	(*****Estop*****)
	IF NOT bEstop  THEN	
		IF eState <> E_Station.eAborted AND eState <> E_Station.eAborting AND eState <> E_Station.eDisabled THEN
				eState 				:= E_Station.eAborting; 
		END_IF
	END_IF
	
	IF bEstop AND bEmergencyUp THEN
		eState 				:= E_Station.eAborting;
	END_IF

	
	CASE eState OF
	/////////////////////////////	
		E_Station.eDisabled: 					// Stan nieaktywnosci (Stacja wyłączona) 
		
			IF bEnable THEN
				eState 				:= E_Station.ePreparingToReady; 
			END_IF 
			
    /////////////////////////////	    
		E_Station.eAborted: 					// Stan bezpiecznego zatrzymania (po Abortingu) 

			IF bEStop THEN
				eState 				:= E_Station.ePreparingToReady;
			END_IF
			
	/////////////////////////////	
		E_Station.eAborting:                 	// Stan bezpiecznego zatrzymywania (po EStopie)
			IF NOT bEstop THEN 
				bBlockActuator 			:= FALSE;
				bLidSealingActuator		:=	FALSE;
				bHeightMotorDown		:=	FALSE;
				bHeightMotorUp			:=	FALSE;
				eState 					:=	E_Station.eAborted;  
				eRunningState			:=	E_LidSealing.eDisabled;
				
			ELSIF bEmergencyUp THEN
								
				bHeightMotorUp			:= NOT tofHeightMotorDown.Q ;
				bHeightMotorDown		:= FALSE;
				bLidSealingActuator		:= FALSE;
				bHomingDone 			:= FALSE;
				IF tonHeightNoChange.Q THEN	
					bHeightMotorEncoderCounterReset	:= TRUE;
					bHeightMotorUp					:= FALSE;
   				END_IF
				
			END_IF
		 
	/////////////////////////////			
		E_Station.eError:                 	 	// Stan błędu 	
			bBlockActuator := FALSE;
			IF bReset THEN
				eState 				:= E_Station.eResetting;
				
			END_IF
			
	/////////////////////////////
		E_Station.eResetting:					// Stan resetowania bledu (po Errorze)
			
			bError := FALSE;
			IF NOT bError THEN
				nErrorNr 			:=	0;
   				sErrorDescription 	:=	'';
				sErrorDescription2	:=	'';
				bTempRegulatorReset := FALSE;
				eState 				:=	E_Station.ePreparingToReady;
			ELSE
				eState 				:=	E_Station.eError;
			END_IF
        
	/////////////////////////////
		E_Station.eManualMovement:     			// Stan ruchów manualnych  
       
			ManualMovements();
			//Wyjście z trybu serwisowego
			IF NOT bManualMovement THEN
				bLidSealingActuator			:=	FALSE;
				bHeightMotorUp				:=	FALSE;
				bHeightMotorDown			:=	FALSE;
				bManualLidSealingActuator	:=	bLidSealingActuator;
				eState:=E_Station.eReady;
			END_IF

	/////////////////////////////
		E_Station.eHoming:						// Stan bazowania 

			Homing();
			IF NOT bHoming AND NOT bHeightSet THEN
			   	eState:=E_Station.ePreparingToReady;
			  	bHeightMotorDown:=FALSE;
				bHeightMotorUp:=FALSE;
			END_IF		
			
	/////////////////////////////
		E_Station.eHomingDone:                  // Stan wykonania bazowania 
		
			bHeightMotorDown					:=	FALSE;
			bHeightMotorUp						:=	FALSE;
			bHeightMotorEncoderCounterReset		:=	FALSE;
			bHomingDone							:=	TRUE;
			IF NOT bHoming AND NOT bHeightSet THEN
			  	 eState:=E_Station.eReady;
			END_IF
			
	/////////////////////////////
		E_Station.ePreparingToReady:            // Stan przygotowywania do gotowosci (zawsze przed Ready)  
		
         	bLidSealingActuator:=FALSE;
			eRunningState:=E_LidSealing.eReady;
			eState:=E_Station.eReady;	
			
	/////////////////////////////
		E_Station.ePreparingToDisable:          // Stan przygotowywania do nieaktywnosci (po wyłączeniu Enable) 
  
			bLidSealingActuator:=FALSE;
			
			bHeightMotorUp:=TRUE;
			bHeightMotorDown:=FALSE;	
			IF tonHeightNoChange.Q THEN
				bHeightMotorUp:=FALSE;
				eState:=E_Station.eDisabled;
				eRunningState:=E_LidSealing.eDisabled;
			END_IF	
			
			
	/////////////////////////////
		E_Station.eReady:						// Stan gotowosci 
		
			IF bRun AND NOT bCycleDone AND NOT bCycleNotDone THEN
				eState 				:= E_Station.eStarting; 
			END_IF
			IF bHoming OR bHeightSet THEN
				eState 				:= E_Station.eHoming; 
			END_IF
			IF bManualMovement THEN
				//Jeśli przejście w tryb ruchów manualnych przepisz wszystkie stany siłowników sterowanych przez moduł
				//aby zapobiec ewentualnym kolizjom po wejściu w tryb serwisowy
				bManualLidSealingActuator	:= bLidSealingActuator;
				bManualHeightMotorUp		:= bHeightMotorUp;
				bManualHeightMotorDown		:= bHeightMotorDown;
				bBlockActuator				:= FALSE;
				eState 						:= E_Station.eManualMovement; 
			END_IF
			IF NOT bRun THEN
				bCycleDone 					:= FALSE;
				bCycleNotDone 				:= FALSE;			
			END_IF
			
	/////////////////////////////
		E_Station.eStopping:					// Stan zatrzymywania 
			
			Running();
			eState 					:= E_Station.eReady;	
			
	/////////////////////////////
		E_Station.eStarting:                  	// Stan uruchamiania (po Ready)
		
			eState					 := E_Station.eRunning; 
			
	/////////////////////////////
		E_Station.eRunning:               		// Stan wykonywania cyklu (po Startingu), w tym stanie osobny
 
			Running();
			IF NOT bRun THEN					(*Przerywanie cyklu*)
				eState 				 := E_Station.eStopping;	
			END_IF
			IF bCycleDone OR bCycleNotDone THEN (*Cykl zakończony*)
				eState 				 := E_Station.eReady;
			END_IF	
			
	/////////////////////////////		
	END_CASE
END_ACTION

ACTION EncoderTest:


rtbHeightMotorEncoderPulse(CLK:=bHeightMotorEncoderPulse,Q=>);
ftbHeightMotorEncoderPulse(CLK:=bHeightMotorEncoderPulse,Q=>);


IF rtbHeightMotorEncoderPulse.Q THEN
	lrHeightMotorEncoderPulses	:=	lrHeightMotorEncoderPulses +	1;
END_IF
END_ACTION

ACTION ErrorHandling:
//OBSŁUGA BŁĘDÓW
// Alarm_0380	380	Error	Blokada siłownika podczas podnoszenia - sprawdź czujnik
// Alarm_0381	381	Error	Blokada siłownika podczas opuszczania - sprawdź czujnik
// Alarm_0382	382	Error	Błąd czujnika temperatury grzałki - sprawdź połączenie
// Alarm_0383	383	Error	Blokada podnośnika lub brak zasilania - sprawdź czujnik lub odblokuj mechanicznie
// Alarm_0384	384	Error	Wartość zadana wysokości jest większa od maksymalnej - zmień ustawienia w recepturze
// Alarm_0385	385	Error	Wartość zadana wysokości jest mniejsza od minimalnej - zmień ustawienia w recepturze
// Alarm_0386	386	Error	Błąd grzania, brak wzrostu temperatury - sprawdź czujnik
// Alarm_0387	387	Error	Błąd grzania, brak sygnału z czujnika temperatury - sprawdź czujnik

IF bAlarmInit THEN
    bAlarmInit := FALSE; 
	fbSourceInfo.Clear();
	fbSourceInfo.sName:=sStationName;//'Machine';
	fbSourceInfo.nId:=udiStationID;//2700;
	// Alarm_0380	380	Error	Blokada siłownika podczas podnoszenia - sprawdź czujnik
    arfbAlarm[0].CreateEx(stEventEntry := TC_EVENTS.AlarmClass.Alarm_0380, bWithConfirmation:= FALSE,  ipSourceInfo:= fbSourceInfo); 
	// Alarm_0381	381	Error	Blokada siłownika podczas opuszczania - sprawdź czujnik
	arfbAlarm[1].CreateEx(stEventEntry := TC_EVENTS.AlarmClass.Alarm_0381, bWithConfirmation:= FALSE,  ipSourceInfo:= fbSourceInfo); 
	// Alarm_0382	382	Error	Błąd czujnika temperatury grzałki - sprawdź połączenie
	arfbAlarm[2].CreateEx(stEventEntry := TC_EVENTS.AlarmClass.Alarm_0382, bWithConfirmation:= FALSE,  ipSourceInfo:= fbSourceInfo); 
	// Alarm_0383	383	Error	Blokada podnośnika lub brak zasilania - sprawdź czujnik lub odblokuj mechanicznie
	arfbAlarm[3].CreateEx(stEventEntry := TC_EVENTS.AlarmClass.Alarm_0383, bWithConfirmation:= FALSE,  ipSourceInfo:= fbSourceInfo); 
	// Alarm_0384	384	Error	Wartość zadana wysokości jest większa od maksymalnej - zmień ustawienia w recepturze
	arfbAlarm[4].CreateEx(stEventEntry := TC_EVENTS.AlarmClass.Alarm_0384, bWithConfirmation:= FALSE,  ipSourceInfo:= fbSourceInfo); 
	// Alarm_0385	385	Error	Wartość zadana wysokości jest mniejsza od minimalnej - zmień ustawienia w recepturze
	arfbAlarm[5].CreateEx(stEventEntry := TC_EVENTS.AlarmClass.Alarm_0385, bWithConfirmation:= FALSE,  ipSourceInfo:= fbSourceInfo); 
	// Alarm_0386	386	Error	Błąd grzania, brak wzrostu temperatury - sprawdź czujnik
	arfbAlarm[6].CreateEx(stEventEntry := TC_EVENTS.AlarmClass.Alarm_0386, bWithConfirmation:= FALSE,  ipSourceInfo:= fbSourceInfo); 
	// Alarm_0387	387	Error	Błąd grzania, brak sygnału z czujnika temperatury - sprawdź czujnik
	arfbAlarm[7].CreateEx(stEventEntry := TC_EVENTS.AlarmClass.Alarm_0387, bWithConfirmation:= FALSE,  ipSourceInfo:= fbSourceInfo); 
END_IF


//GRZAŁKI NIEGOTOWE (różnica temperatury grzałki różna od zadanej +/-10 st.C 
IF (ABS(lrHeaterTemperatureCVSensor-nHeaterTemperatureSV)>nTempHisteresis AND NOT bHeaterTemperatureErrorIgnore) AND eRunningState=E_LidSealing.eReady THEN
		eRunningState:=E_LidSealing.eHeaterNotReady;		
ELSIF eRunningState=E_LidSealing.eHeaterNotReady THEN
		IF (ABS(lrHeaterTemperatureCVSensor-nHeaterTemperatureSV)<nTempHisteresis OR bHeaterTemperatureErrorIgnore) THEN
			eRunningState:=E_LidSealing.eReady;	
		END_IF	
END_IF


//************LISTA BŁĘDÓW***************
bStateError:= (eState=E_Station.eError) OR (eState=E_Station.eResetting) OR bIgnoreError;


IF bEnable THEN
	// Alarm_0380	380	Error	Blokada siłownika podczas podnoszenia - sprawdź czujnik
	//Error 1 - Zacięcie siłownika zgrzewania przy próbie podnoszenia
	tonSealingActuatorUpLag(IN:=NOT bLidSealingActuator AND NOT bLidSealingActuatorUpSensor,PT:=T#2S);
	IF tonSealingActuatorUpLag.Q THEN
		IF NOT arfbAlarm[0].bActive THEN
			bLidSealingActuator:=FALSE;
			arfbAlarm[0].Raise(nTimeStamp:=0);
		END_IF
	ELSE	
		IF  arfbAlarm[0].bActive AND bReset THEN
			arfbAlarm[0].Clear(nTimeStamp:=0, bResetConfirmation:= FALSE);
		END_IF	
// 		bLidSealingActuator:=FALSE;
// 		bError := TRUE;
// 		nErrorNr:=251;
// 		//nErrorNr := nErrorNr+iStationIndex;
// 		sErrorDescription:='Blokada siłownika podczas podnoszenia - sprawdź czujnik';
	END_IF;
	// Alarm_0381	381	Error	Blokada siłownika podczas opuszczania - sprawdź czujnik
	//Error 2 - Zacięcie siłownika zgrzewania przy próbie opuszczania
	tonSealingActuatorDownLag(IN:=bLidSealingActuator AND NOT bLidSealingActuatorDownSensor,PT:=T#2S);
	IF tonSealingActuatorDownLag.Q THEN
		IF NOT arfbAlarm[1].bActive THEN
			bLidSealingActuator:=FALSE;
			arfbAlarm[1].Raise(nTimeStamp:=0);
		END_IF
	ELSE	
		IF  arfbAlarm[1].bActive AND bReset THEN
			arfbAlarm[1].Clear(nTimeStamp:=0, bResetConfirmation:= FALSE);
		END_IF	
// 		bLidSealingActuator:=FALSE;
// 		bError := TRUE;
// 		nErrorNr:=252;
// 		//nErrorNr := nErrorNr+iStationIndex;
// 		sErrorDescription:='Blokada siłownika podczas opuszczania - sprawdź czujnik';	
	END_IF;
	// Alarm_0382	382	Error	Błąd czujnika temperatury grzałki - sprawdź połączenie
	//Error 3 - Błąd czujnika temperatury
	IF bHeaterEnable AND bTemperatureSensorFault THEN
		IF NOT arfbAlarm[2].bActive THEN
			arfbAlarm[2].Raise(nTimeStamp:=0);
			bTempRegulatorReset:=TRUE;
		END_IF
	ELSE	
		IF  arfbAlarm[2].bActive AND bReset THEN
			arfbAlarm[2].Clear(nTimeStamp:=0, bResetConfirmation:= FALSE);
		END_IF	
//		bTempRegulatorReset:=TRUE;
// 		bError := TRUE;
// 		nErrorNr:=253;
// 		//nErrorNr := nErrorNr+iStationIndex;
// 		sErrorDescription:='Błąd czujnika temperatury grzałki - sprawdź połączenie';	
	END_IF;
	// Alarm_0383	383	Error	Blokada podnośnika lub brak zasilania - sprawdź czujnik lub odblokuj mechanicznie
	//Error 4 - podnośnik nie porusza się pomimo wysterowania 
	tonErrorHeightChange(IN:=(bHeightMotorUp OR bHeightMotorDown) AND nLastPositionHeightCV=lrHeightMotorCV, PT:=T#3S);
	IF tonErrorHeightChange.Q THEN
		IF NOT arfbAlarm[3].bActive THEN
			arfbAlarm[3].Raise(nTimeStamp:=0);
			bHeightMotorUp:=FALSE;
			bHeightMotorDown:=FALSE;
		END_IF
	ELSE	
		IF  arfbAlarm[3].bActive AND bReset THEN
			arfbAlarm[3].Clear(nTimeStamp:=0, bResetConfirmation:= FALSE);
		END_IF	
// 		bHeightMotorUp:=FALSE;
// 		bHeightMotorDown:=FALSE;
// 		bError := TRUE;
// 		nErrorNr:=254;
// 		//nErrorNr := nErrorNr+iStationIndex;
// 		sErrorDescription:='Blokada podnośnika lub brak zasilania - sprawdź czujnik lub odblokuj mechanicznie';	
	END_IF
	// Alarm_0384	384	Error	Wartość zadana wysokości jest większa od maksymalnej - zmień ustawienia w recepturze
	//Error 5 - Bład nastaw max
	tonMaxHeight(IN:=nPositionHeightSV>lrMaxHeight AND NOT bHomingDone AND eState=E_Station.eReady,PT:=T#30S);
	IF tonMaxHeight.Q THEN
		arfbAlarm[4].ipArguments.Clear() .AddLReal(lrMaxHeight);
		IF NOT arfbAlarm[4].bActive THEN
			bHeightMotorUp:=FALSE;
			bHeightMotorDown:=FALSE;
			arfbAlarm[4].Raise(nTimeStamp:=0);
		END_IF
	ELSE	
		IF  arfbAlarm[4].bActive AND bReset THEN
			arfbAlarm[4].Clear(nTimeStamp:=0, bResetConfirmation:= FALSE);
		END_IF	
// 		bHeightMotorUp:=FALSE;
// 		bHeightMotorDown:=FALSE;
// 		bError := TRUE;
// 		nErrorNr:=255;
// 		//nErrorNr := nErrorNr+iStationIndex;
// 		sErrorDescription:='Wartość zadana wysokości jest większa od maksymalnej - zmień ustawienia w recepturze';
// 		sErrorDescription2:=REAL_TO_STRING(LREAL_TO_INT(lrMaxHeight));
	END_IF
	// Alarm_0385	385	Error	Wartość zadana wysokości jest mniejsza od minimalnej - zmień ustawienia w recepturze
	//Error 6 - Bład nastaw min
	tonMinHeight(IN:=nPositionHeightSV<lrMinHeight AND NOT bHomingDone AND eState=E_Station.eReady,PT:=T#30S);
	IF tonMinHeight.Q THEN
		arfbAlarm[5].ipArguments.Clear() .AddLReal(lrMinHeight);
		IF NOT arfbAlarm[5].bActive THEN
			bHeightMotorUp:=FALSE;
			bHeightMotorDown:=FALSE;
			arfbAlarm[5].Raise(nTimeStamp:=0);
		END_IF
	ELSE	
		IF  arfbAlarm[5].bActive AND bReset THEN
			arfbAlarm[5].Clear(nTimeStamp:=0, bResetConfirmation:= FALSE);
		END_IF	
// 		bHeightMotorUp:=FALSE;
// 		bHeightMotorDown:=FALSE;
// 		bError := TRUE;
// 		nErrorNr:=256;
// 		//nErrorNr := nErrorNr+iStationIndex;
// 		sErrorDescription:='Wartość zadana wysokości jest mniejsza od minimalnej - zmień ustawienia w recepturze';
// 		sErrorDescription2:=REAL_TO_STRING(LREAL_TO_INT(lrMinHeight));	
	END_IF
	// Alarm_0386	386	Error	Błąd grzania, brak wzrostu temperatury - sprawdź czujnik
	//Error 7 - Błąd czujnika temperatury
	tofbHeaterPWMOut(IN:=bHeaterPWMOut,PT:=T#30S);
	tonHeaterOnAndNotHeating(IN:=tofbHeaterPWMOut.Q AND lrHeaterTemperatureCVSensor=lrHeaterTemperatureCVSensorLast AND NOT bIgnoreError , PT:=T#5M);
	lrHeaterTemperatureCVSensorLast := lrHeaterTemperatureCVSensor;
	IF tonHeaterOnAndNotHeating.Q THEN
		IF NOT arfbAlarm[6].bActive THEN
			bTempRegulatorReset 	:= TRUE;
			arfbAlarm[6].Raise(nTimeStamp:=0);
		END_IF
	ELSE	
		IF  arfbAlarm[6].bActive AND bReset THEN
			arfbAlarm[6].Clear(nTimeStamp:=0, bResetConfirmation:= FALSE);
		END_IF	
//  		bTempRegulatorReset 	:= TRUE;
// 		bError 					:= TRUE;
// 		nErrorNr 				:= 257;
// 		//nErrorNr				:=nErrorNr+iStationIndex;
// 		sErrorDescription 		:= 'Błąd grzania, brak wzrostu temperatury - sprawdź czujnik';	
	END_IF
	// Alarm_0387	387	Error	Błąd grzania, brak sygnału z czujnika temperatury - sprawdź czujnik
	//Error 8 - Błąd czujnika temperatury, wskazuje 0
	tonHeaterOnAndSensorShows0(IN:=bHeaterPWMOut AND lrHeaterTemperatureCVSensor<1 AND NOT bIgnoreError AND NOT bStateError , PT:=T#15S);
	IF tonHeaterOnAndSensorShows0.Q THEN
		IF NOT arfbAlarm[7].bActive THEN
			bTempRegulatorReset 	:= TRUE;
			arfbAlarm[7].Raise(nTimeStamp:=0);
		END_IF
	ELSE	
		IF  arfbAlarm[7].bActive AND bReset THEN
			arfbAlarm[7].Clear(nTimeStamp:=0, bResetConfirmation:= FALSE);
		END_IF	
//  		bTempRegulatorReset 	:= TRUE;
// 		bError 					:= TRUE;
// 		nErrorNr 				:= 258;
// 		//nErrorNr				:=nErrorNr+iStationIndex;
// 		sErrorDescription 		:= 'Błąd grzania, brak sygnału z czujnika temperatury - sprawdź czujnik';	
	END_IF	
	
ELSE
	bError := FALSE;
END_IF

//*******KONIEC LISTA BŁĘDÓW***************
	

//******************PRZEJŚCIE DO eERROR*****************************

IF bError AND NOT bStateError THEN
	IF eLastState = eRunning THEN
		bCycleNotDone := TRUE;
	END_IF
	eState := E_Station.eError;
END_IF

//****************WYŚWIETLANIE STATUSU BLEDU***********************


(*Wyświetlanie błedu na wyjściu*)
bError							:= FALSE;
FOR nAlarmNumerator := 0 TO 19 DO
	bError						:= bError OR arfbAlarm[nAlarmNumerator].bActive;
END_FOR

(*Przepisywanie nazwy stacji*)
sErrorStationName:=sStationName;



//Jezeli nie zbazowane to potrzebne bazowanie
IF NOT bHeightMotorEncoderHomed  THEN
	bHomingDone:=FALSE;
END_IF
END_ACTION

ACTION HeaterRegulator:
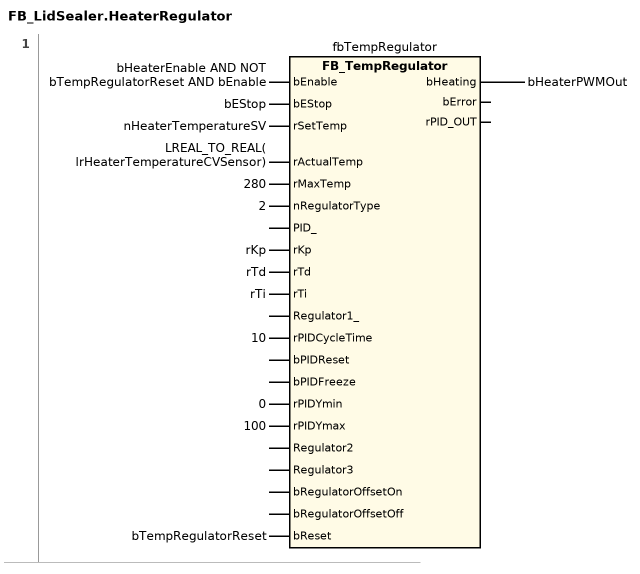
// NETWORK 1
fbTempRegulator(
    bEnable := bHeaterEnable AND NOT bTempRegulatorReset AND bEnable,
    bEStop := bEStop,
    rSetTemp := nHeaterTemperatureSV,
    rActualTemp := LREAL_TO_REAL(lrHeaterTemperatureCVSensor),
    rMaxTemp := 280,
    nRegulatorType := 2,
    rKp := rKp,
    rTd := rTd,
    rTi := rTi,
    rPIDCycleTime := 10,
    rPIDYmin := 0,
    rPIDYmax := 100,
    bReset := bTempRegulatorReset); // FB_TempRegulator
bHeaterPWMOut := fbTempRegulator.bHeating;
END_ACTION

ACTION HeightMotor:
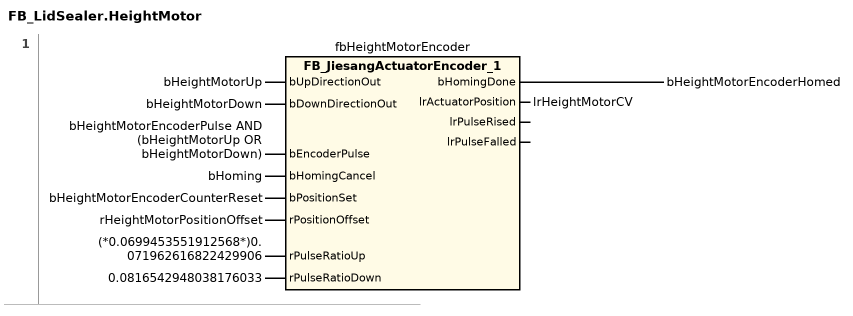
// NETWORK 1
fbHeightMotorEncoder(
    bUpDirectionOut := bHeightMotorUp,
    bDownDirectionOut := bHeightMotorDown,
    bEncoderPulse := bHeightMotorEncoderPulse AND (bHeightMotorUp OR bHeightMotorDown),
    bHomingCancel := bHoming,
    bPositionSet := bHeightMotorEncoderCounterReset,
    rPositionOffset := rHeightMotorPositionOffset,
    rPulseRatioUp := (*0.0699453551912568*)0.071962616822429906,
    rPulseRatioDown := 0.0816542948038176033,
    lrActuatorPosition => lrHeightMotorCV); // FB_JiesangActuatorEncoder_1
bHeightMotorEncoderHomed := fbHeightMotorEncoder.bHomingDone;
END_ACTION

ACTION Homing:
//BAZOWANIE
bLidSealingActuator:=FALSE;
//tofHeightMotorDown(IN:=bHeightMotorDown, PT:=T#1S); //Zabezpieczenie przed zbyt szybkim przełączeniem pomiędzy Down a Up, bezpiecznieki sie palą
		
//Podnoszenie stacji do maksymalnej pozycji
IF NOT bHeightMotorEncoderHomed OR rtEncoderHomed.Q THEN
	bHeightMotorUp:=(*TRUE*) NOT tofHeightMotorDown.Q ;
	bHeightMotorDown:=FALSE;
	IF tonHeightNoChange.Q THEN
		bHeightMotorEncoderCounterReset:=TRUE;
		bHeightMotorUp:=FALSE;
    END_IF
	//Jesli enkoder zbazowany zakończ bazowanie	
	IF rtEncoderHomed.Q THEN
		bHeightMotorUp:=FALSE;
		bHeightMotorDown:=FALSE;
		eState:=E_Station.eHomingDone;
	END_IF		
		
//Po podniesieniu stacji opuszczanie do ustalonej wysokości
ELSIF bHeightMotorEncoderHomed THEN
	bHeightMotorEncoderCounterReset:=FALSE;
	bHeightMotorUp:=lrHeightMotorCV<=nPositionHeightSV;
	bHeightMotorDown:=lrHeightMotorCV>=nPositionHeightSV;
	//Kiedy stacja osiągnie wysokość zadaną
	IF ABS(lrHeightMotorCV-nPositionHeightSV)<1 OR tonLimitPosMaxReachedDelay.Q OR tonLimitPosMinReachedDelay.Q THEN
		bHeightMotorDown:=FALSE;
		bHeightMotorUp:=FALSE;
		eState:=E_Station.eHomingDone;
	END_IF			
END_IF
END_ACTION

ACTION ManualMovements:

//W trybie ruchów manualnych wykonuj ruchy za pomocą rozkazów manualnych
IF NOT bRun THEN
	
	bBlockActuator:=bManualLidSealingActuator;
	bLidSealingActuator:=tonbBlockActuator.Q;
	bHeightMotorUp:=bManualHeightMotorUp;
	bHeightMotorDown:=bManualHeightMotorDown;
ELSE	//Kasuje zeby po cyklu nic sie nie poruszało
	bManualLidSealingActuator := FALSE;
	bManualHeightMotorUp  := FALSE;
	bManualHeightMotorDown  := FALSE;
END_IF


IF bHoming OR bHeightSet THEN
	eState:=E_Station.eHoming;
END_IF
	
Running();
	
//Zabezpieczenie przed kolizją stacji poprzez ruch podnośnika	
IF bHeightMotorDown AND lrHeightMotorCV<=lrMinHeight AND NOT bHoming AND NOT bHeightSet THEN
	bHeightMotorDown:=FALSE;
END_IF	

IF bHeightMotorUp AND lrHeightMotorCV>=lrMaxHeight AND NOT bHoming AND NOT bHeightSet THEN
	bHeightMotorUp:=FALSE;
END_IF		 

IF NOT bRun THEN
	bCycleDone 					:= FALSE;
	bCycleNotDone 				:= FALSE;	
END_IF
END_ACTION

ACTION Protections:
(*Nadpisywanie sygnałów dla bezpieczństwa mechaniki*)
IF bHeightMotorDisable THEN // Włączony siłownik blokujący podnoszenie
	bHeightMotorUp		:=FALSE;	
	bHeightMotorDown	:=FALSE;	
END_IF
END_ACTION

ACTION Running:

//Timery 
tonHeatingTime(IN:=eRunningState=E_LidSealing.eHeating,PT:=INT_TO_TIME(nLidHeatingTime));
tonbNOTLidSealingActuator(IN:=NOT bLidSealingActuator AND eRunningState=E_LidSealing.eHeating, PT:=T#100MS);
tonbBlockActuator(IN:=bBlockActuator,PT:=T#400MS);

CASE eRunningState OF
	
	//NIEGOTOWY
	E_LidSealing.eDisabled:
			eRunningState:=E_LidSealing.eReady;
		
	//ZGRZEWANIE GOTOWY DO PRACY
	E_LidSealing.eReady:
		//bLidSealingActuator:=FALSE;
		//Jeśli komenda podania platynki przejdź do stanu zasysania platynki
		IF NOT bCycleDone AND NOT bCycleNotDone THEN
			IF bRun THEN
				IF NOT bManualMovement THEN
					eRunningState:=E_LidSealing.eSealing;
				ELSE
					bBlockActuator := TRUE;
					IF tonbBlockActuator.Q THEN
						eRunningState:=E_LidSealing.eSealing;
					END_IF
				END_IF
			END_IF
		END_IF

	//STAN ZGRZEWANIA - opuszaczanie siłownika grzałki
	E_LidSealing.eSealing:
		bLidSealingActuator:=TRUE;
		//Jeśli komenda podania platynki przejdź do stanu opuszczania siłownika podajnika
		IF bLidSealingActuatorDownSensor THEN
			eRunningState:=E_LidSealing.eHeating;
		END_IF

	//ZGRZEWANIE PLATYNKI
	E_LidSealing.eHeating:
		//Zgrzewanie platynki dopóki nie osiągnie czasu przygrzewania
		IF NOT tonHeatingTime.Q THEN
			bLidSealingActuator:=TRUE;
		ELSE
			bLidSealingActuator:=FALSE;
			//IF NOT bLidSealingActuatorUpSensor THEN
			IF 	tonbNOTLidSealingActuator.Q THEN
				eRunningState:=E_LidSealing.eLidSealed;	
			END_IF
		END_IF
	
	//Zgrzewanie zakończone
	E_LidSealing.eLidSealed:
	
		bLidSealingActuator := FALSE;
		bCycleDone := TRUE;
		IF bLidSealingActuatorUpSensor THEN
			eRunningState:=E_LidSealing.eReady;
		ELSE
			eRunningState:=E_LidSealing.eGoingUp;
		END_IF

	//PODAJNIK PODNOSI SIŁOWNIK PODAWANIA PLATYNEK
	E_LidSealing.eGoingUp:
		bLidSealingActuator:=FALSE;
		bBlockActuator := FALSE;
		IF bLidSealingActuatorUpSensor THEN
			eRunningState:=E_LidSealing.eReady;
		END_IF

END_CASE
END_ACTION

ACTION Statistics:

rtrigCycleTimerRead(CLK:=(eRunningState=E_LidSealing.eLidSealed));
IF rtrigCycleTimerRead.Q THEN
		tCycleTime:=tonCycleTimer.ET;
END_IF
tonCycleTimer(IN:=eRunningState>E_LidSealing.eReady,PT:=T#1D);
END_ACTION

END_FUNCTION_BLOCK

// ---- POUs/P00_ReadRFIDCard.TcPOU
(*
Nazwa:			P00_ReadRFIDCard
Opis:			Czytnik kart zbliżeniowych
Wersja:			v0.12
Data:			2022-02-07
Autor:			DP
Urzadzenia:		
Konfiguracja:	
Info:
- Przerobienie programu na nowe czujniki RFID IFM'a
- Programować formatki trzeba po staremu bo ten bloczek IFMa nie przetestowany
*)
PROGRAM P00_ReadRFIDCard
VAR



	bReadedCardDispencer :BOOL;					(*PLC.A10*)		//Wykrycie nośnika przez czytnik przy dozownikach	
	bReadedCardBeforeScrewer :BOOL;				(*PLC.A10*)		//Wykrycie nośnika przez czytnik na 1 wjeździe karuzeli
	bReadedCardAfterScrewer :BOOL;				(*PLC.A10*)		//Wykrycie nośnika przez czytnik na 1 wjeździe karuzeli
	bReadedCardAfterDispencers :BOOL;			(*PLC.A10*)		//Wykrycie nośnika przez czytnik na 2 wjeździe karuzeli
	bReadedCardBottleTransfer :BOOL;			(*PLC.A10*)		//Wykrycie nośnika przez czytnik przy robocie
	bReadedCardCapSorter :BOOL;					(*PLC.A10*)		//Wykrycie nośnika przez czytnik przy robocie
	bReadedCardAfterDispencers2Phase :BOOL;		(*PLC.A10*)		//Wykrycie nośnika przez czytnik przy robocie
	bReadedCardLidFeeder :BOOL;					(*PLC.A10*)		//Wykrycie nośnika przez czytnik na 1 wjeździe karuzeli
	bReadedCardLidSealer :BOOL;
	
	nReadedCardDispencer :ULINT;								
	nReadedCardBeforeScrewer :ULINT;							
	nReadedCardAfterScrewer	:ULINT;
	nReadedCardAfterDispencers :ULINT;							
	nReadedCardBottleTransfer :ULINT;			
	nReadedCardCapSorter :ULINT;	
	nReadedCardAfterDispencers2Phase :ULINT;	
	nReadedCardLidFeeder :ULINT;
	nReadedCardLidSealer :ULINT;	
			
	fbWriteDataRFID: FB_WriteRFID;
	fbWriteDataRFIDnew: FB_WriteRFIDnew;
	bAutoNumber: BOOL;
	byIDtoWrite: BYTE;
	bReset: BOOL;
	bE: BOOL;
	
	(*Nowa Głowica IFM*)
	fbDispencerReader   								:   	FB_IfmIoLinkRfid;
	AusiDispencerReaderInputData  				AT%I*	: 		ARRAY[0..27] OF USINT;
	IbDispencerReaderTagPresent					AT%I*	:		BOOL;
	IBDispencerReaderErrorValue					AT%I*	:		BYTE;
	IbDispencerReaderCmdEnd						AT%I*	:		BOOL;
	IBDispencerReaderDataCounterIn				AT%I*	:		BYTE;
	IbDispencerReaderCmdStartAck				AT%I*	:		BOOL;
	IbDispencerReaderCmdStart					AT%Q*	:		BOOL;
	IBDispencerReaderCmmandValue				AT%Q*	:		BYTE;
	IBDispencerReaderDataCounterOut				AT%Q*	:		BYTE;
	AusiDispencerReaderOutputData  				AT%Q*	: 		ARRAY[0..27] OF USINT;	
	
	fbAfterDispencersReader   							:   	FB_IfmIoLinkRfid;
	AusiAfterDispencersReaderInputData  		AT%I*	: 		ARRAY[0..27] OF USINT;
	IbAfterDispencersReaderTagPresent			AT%I*	:		BOOL;
	IBAfterDispencersReaderErrorValue			AT%I*	:		BYTE;
	IbAfterDispencersReaderCmdEnd				AT%I*	:		BOOL;
	IBAfterDispencersReaderDataCounterIn		AT%I*	:		BYTE;
	IbAfterDispencersReaderCmdStartAck			AT%I*	:		BOOL;
	IbAfterDispencersReaderCmdStart				AT%Q*	:		BOOL;
	IBAfterDispencersReaderCmmandValue			AT%Q*	:		BYTE;
	IBAfterDispencersReaderDataCounterOut		AT%Q*	:		BYTE;
	AusiAfterDispencersReaderOutputData  		AT%Q*	: 		ARRAY[0..27] OF USINT;		
	ABAfterDispencersReaderWriteData					:		ARRAY[0..15] OF BYTE;

	fbLidFeederReader   								:   	FB_IfmIoLinkRfid; 	
	AusiLidFeederReaderInputData  				AT%I*	: 		ARRAY[0..27] OF USINT;
	IbLidFeederReaderTagPresent					AT%I*	:		BOOL;
	IBLidFeederReaderErrorValue					AT%I*	:		BYTE;
	IbLidFeederReaderCmdEnd						AT%I*	:		BOOL;
	IBLidFeederReaderDataCounterIn				AT%I*	:		BYTE;
	IbLidFeederReaderCmdStartAck				AT%I*	:		BOOL;
	IbLidFeederReaderCmdStart					AT%Q*	:		BOOL;
	IBLidFeederReaderCmmandValue				AT%Q*	:		BYTE;
	IBLidFeederReaderDataCounterOut				AT%Q*	:		BYTE;
	AusiLidFeederReaderOutputData  				AT%Q*	: 		ARRAY[0..27] OF USINT;		
	ABALidFeederReaderWriteData							:		ARRAY[0..15] OF BYTE;
	
	fbBeforeScrewerReader   							:   	FB_IfmIoLinkRfid;
	AusiBeforeScrewerReaderInputData  			AT%I*	: 		ARRAY[0..27] OF USINT;
	IbBeforeScrewerReaderTagPresent				AT%I*	:		BOOL;
	IBBeforeScrewerReaderErrorValue				AT%I*	:		BYTE;
	IbBeforeScrewerReaderCmdEnd					AT%I*	:		BOOL;
	IBBeforeScrewerReaderDataCounterIn			AT%I*	:		BYTE;
	IbBeforeScrewerReaderCmdStartAck			AT%I*	:		BOOL;
	IbBeforeScrewerReaderCmdStart				AT%Q*	:		BOOL;
	IBBeforeScrewerReaderCmmandValue			AT%Q*	:		BYTE;
	IBBeforeScrewerReaderDataCounterOut			AT%Q*	:		BYTE;
	AusiBeforeScrewerReaderOutputData  			AT%Q*	: 		ARRAY[0..27] OF USINT;	

	fbAfterScrewerReader   								:   	FB_IfmIoLinkRfid;
	AusiAfterScrewerReaderInputData  			AT%I*	: 		ARRAY[0..27] OF USINT;
	IbAfterScrewerReaderTagPresent				AT%I*	:		BOOL;
	IBAfterScrewerReaderErrorValue				AT%I*	:		BYTE;
	IbAfterScrewerReaderCmdEnd					AT%I*	:		BOOL;
	IBAfterScrewerReaderDataCounterIn			AT%I*	:		BYTE;
	IbAfterScrewerReaderCmdStartAck				AT%I*	:		BOOL;
	IbAfterScrewerReaderCmdStart				AT%Q*	:		BOOL;
	IBAfterScrewerReaderCmmandValue				AT%Q*	:		BYTE;
	IBAfterScrewerReaderDataCounterOut			AT%Q*	:		BYTE;
	AusiAfterScrewerReaderOutputData  			AT%Q*	: 		ARRAY[0..27] OF USINT;	

	fbBottleTransferReader   							:   	FB_IfmIoLinkRfid;
	AusiBottleTransferReaderInputData  			AT%I*	: 		ARRAY[0..27] OF USINT;
	IbBottleTransferReaderTagPresent			AT%I*	:		BOOL;
	IBBottleTransferReaderErrorValue			AT%I*	:		BYTE;
	IbBottleTransferReaderCmdEnd				AT%I*	:		BOOL;
	IBBottleTransferReaderDataCounterIn			AT%I*	:		BYTE;
	IbBottleTransferReaderCmdStartAck			AT%I*	:		BOOL;
	IbBottleTransferReaderCmdStart				AT%Q*	:		BOOL;
	IBBottleTransferReaderCmmandValue			AT%Q*	:		BYTE;
	IBBottleTransferReaderDataCounterOut		AT%Q*	:		BYTE;
	AusiBottleTransferReaderOutputData  		AT%Q*	: 		ARRAY[0..27] OF USINT;		
	
	fbCapSorterReader   								:   	FB_IfmIoLinkRfid;
	AusiCapSorterReaderInputData  				AT%I*	: 		ARRAY[0..27] OF USINT;
	IbCapSorterReaderTagPresent					AT%I*	:		BOOL;
	IBCapSorterReaderErrorValue					AT%I*	:		BYTE;
	IbCapSorterReaderCmdEnd						AT%I*	:		BOOL;
	IBCapSorterReaderDataCounterIn				AT%I*	:		BYTE;
	IbCapSorterReaderCmdStartAck				AT%I*	:		BOOL;
	IbCapSorterReaderCmdStart					AT%Q*	:		BOOL;
	IBCapSorterReaderCmmandValue				AT%Q*	:		BYTE;
	IBCapSorterReaderDataCounterOut				AT%Q*	:		BYTE;
	AusiCapSorterReaderOutputData  				AT%Q*	: 		ARRAY[0..27] OF USINT;		
	
	fbAfterDispencers2PhaseReader   						:   	FB_IfmIoLinkRfid;
	AusiAfterDispencers2PhaseReaderInputData  		AT%I*	: 		ARRAY[0..27] OF USINT;
	IbAfterDispencers2PhaseReaderTagPresent			AT%I*	:		BOOL;
	IBAfterDispencers2PhaseReaderErrorValue			AT%I*	:		BYTE;
	IbAfterDispencers2PhaseReaderCmdEnd				AT%I*	:		BOOL;
	IBAfterDispencers2PhaseReaderDataCounterIn		AT%I*	:		BYTE;
	IbAfterDispencers2PhaseReaderCmdStartAck		AT%I*	:		BOOL;
	IbAfterDispencers2PhaseReaderCmdStart			AT%Q*	:		BOOL;
	IBAfterDispencers2PhaseReaderCmmandValue		AT%Q*	:		BYTE;
	IBAfterDispencers2PhaseReaderDataCounterOut		AT%Q*	:		BYTE;
	AusiAfterDispencers2PhaseReaderOutputData  		AT%Q*	: 		ARRAY[0..27] OF USINT;		
	ABAfterDispencers2PhaseReaderWriteData					:		ARRAY[0..15] OF BYTE;
	
	fbLidSealerReader   								:   	FB_IfmIoLinkRfid; 	
	AusiLidSealerReaderInputData  				AT%I*	: 		ARRAY[0..27] OF USINT;
	IbLidSealerReaderTagPresent					AT%I*	:		BOOL;
	IBLidSealerReaderErrorValue					AT%I*	:		BYTE;
	IbLidSealerReaderCmdEnd						AT%I*	:		BOOL;
	IBLidSealerReaderDataCounterIn				AT%I*	:		BYTE;
	IbLidSealerReaderCmdStartAck				AT%I*	:		BOOL;
	IbLidSealerReaderCmdStart					AT%Q*	:		BOOL;
	IBLidSealerReaderCmmandValue				AT%Q*	:		BYTE;
	IBLidSealerReaderDataCounterOut				AT%Q*	:		BYTE;
	AusiLidSealerReaderOutputData  				AT%Q*	: 		ARRAY[0..27] OF USINT;	
	ABALidSealerReaderWriteData							:		ARRAY[0..15] OF BYTE;
	
	
	(**)
	iWriteDataCASE										:	INT;
	iWriteDataOn										:	BOOL;
	iWriteDataCount										:	INT;
	tonWriteDataCASE40									:	TON;
	
	(*RFIDCheck*)
	rtbWeighingFormDone									:	R_TRIG;

	
	tonRFIDCheckReader1Add								:	TON;
	rtRFIDCheckReader1Add								:	R_TRIG;
	tonRFIDCheckReader2Add								:	TON;
	rtRFIDCheckReader2Add								:	R_TRIG;
	tonRFIDCheckReader3Add								:	TON;
	rtRFIDCheckReader3Add								:	R_TRIG;
	tonRFIDCheckReader4Add								:	TON;
	rtRFIDCheckReader4Add								:	R_TRIG;
	tonRFIDCheckReader5Add								:	TON;
	rtRFIDCheckReader5Add								:	R_TRIG;	



	//AuliRFIDCheck										:	ARRAY [1..100] OF ULINT;	

	bRFIDCheckSave										:	BOOL;
	iRFIDCheck											:	INT;
	rtRFIDCheckbReadedCardBottleTransfer				:	R_TRIG;
	bRFIDCheckDiffrence									:	BOOL;
	iRFIDCheckProblemWithNumber							:	INT;
	sRFIDInfoSensorError								:	STRING;
	iRFIDCheckNumberOfFormsExecuteTemp					:	INT;	
	i,j													:	INT;
	
	tonRFIDCheckDispencersWarning						:	TON;
	rttonRFIDCheckDispencerWarning						:	R_TRIG;

	iRFIDCheckDispencerWarningLast						:	INT;	
	bRFIDCheckDispencerWarning							:	BOOL;
	
	tonRFIDCheckWeightWarning						:	TON;
	rttonRFIDCheckWeightWarning						:	R_TRIG;

	iRFIDCheckWeightWarningLast						:	INT;
	
	bRFIDCheckWeightWarning							:	BOOL;
	
	tonRFIDCheckBeforeScrewerWarning				:	TON;
	rttonRFIDCheckBeforeScrewerWarning				:	R_TRIG;

	iRFIDCheckBeforeScrewerWarningLast				:	INT;	
	bRFIDCheckBeforeScrewerWarning					:	BOOL;
	
	tonRFIDCheckAfterScrewerWarning					:	TON;
	rttonRFIDCheckAfterScrewerWarning				:	R_TRIG;

	iRFIDCheckAfterScrewerWarningLast				:	INT;
	
	bRFIDCheckAfterScrewerWarning					:	BOOL;	

	tonRFIDCheckBottleTransferWarning				:	TON;
	rttonRFIDCheckBottleTransferWarning				:	R_TRIG;

	iRFIDCheckBottleTransferWarningLast				:	INT;

	bRFIDCheckBottleTransferWarning					:	BOOL;	


	tonRFIDCheck10s									:	TON;
	ftRFIDCheckAfterScrewerWarning					:	F_TRIG;
	bRFIDCheckResetAll								:	BOOL;
	tonRFIDReset									:	TON;
	iRFIDReaded1Errors								: 	INT;
	iRFIDReaded2Errors								: 	INT;
	iRFIDReaded3Errors								: 	INT;
	iRFIDReaded4Errors								: 	INT;
	iRFIDReaded5Errors								: 	INT;	
	bRFIDCheckEnable								:	BOOL;
	
	(*inne*)
	




END_VAR

(*Przepisanie bity wykrycia karty*)
bReadedCardDispencer 		:= IbDispencerReaderTagPresent AND fbDispencerReader.bCodeReaded;
nReadedCardDispencer 		:= DINT_TO_ULINT(P00_ReadRFIDCard.fbDispencerReader.diReadedCode);

bReadedCardAfterDispencers 	:= IbAfterDispencersReaderTagPresent AND fbAfterDispencersReader.bCodeReaded;
nReadedCardAfterDispencers	:= DINT_TO_ULINT(P00_ReadRFIDCard.fbAfterDispencersReader.diReadedCode);

bReadedCardBeforeScrewer 	:= IbBeforeScrewerReaderTagPresent AND fbBeforeScrewerReader.bCodeReaded;
nReadedCardBeforeScrewer	:= DINT_TO_ULINT(P00_ReadRFIDCard.fbBeforeScrewerReader.diReadedCode);

bReadedCardAfterScrewer 	:= IbAfterScrewerReaderTagPresent  AND fbAfterScrewerReader.bCodeReaded;
nReadedCardAfterScrewer		:= DINT_TO_ULINT(P00_ReadRFIDCard.fbAfterScrewerReader.diReadedCode);

bReadedCardBottleTransfer 	:= IbBottleTransferReaderTagPresent AND fbBottleTransferReader.bCodeReaded;;
nReadedCardBottleTransfer	:= DINT_TO_ULINT(P00_ReadRFIDCard.fbBottleTransferReader.diReadedCode);

bReadedCardCapSorter 		:= IbCapSorterReaderTagPresent AND fbCapSorterReader.bCodeReaded;;
nReadedCardCapSorter		:= DINT_TO_ULINT(P00_ReadRFIDCard.fbCapSorterReader.diReadedCode);

bReadedCardAfterDispencers2Phase 	:= IbAfterDispencers2PhaseReaderTagPresent AND fbAfterDispencers2PhaseReader.bCodeReaded;
nReadedCardAfterDispencers2Phase	:= DINT_TO_ULINT(P00_ReadRFIDCard.fbAfterDispencers2PhaseReader.diReadedCode);

bReadedCardLidFeeder 		:= IbLidFeederReaderTagPresent AND fbLidFeederReader.bCodeReaded;;
nReadedCardLidFeeder 		:= DINT_TO_ULINT(P00_ReadRFIDCard.fbLidFeederReader.diReadedCode);

bReadedCardLidSealer 		:= IbLidSealerReaderTagPresent AND fbLidSealerReader.bCodeReaded;;
nReadedCardLidSealer 		:= DINT_TO_ULINT(P00_ReadRFIDCard.fbLidSealerReader.diReadedCode);




aIFM();
aWriteDataIFM();
aHMIShowRFID();
aRFIDCheck();
aRFIDCheckWarnings();

ACTION aHMIShowRFID:

VIS.sSlowestStation5:= Concat('RFID before scales:',ULINT_TO_STRING(nReadedCardAfterDispencers));
VIS.iSlowestStationCount5:=ULINT_TO_INT(nReadedCardAfterDispencers);
END_ACTION

ACTION aIFM:
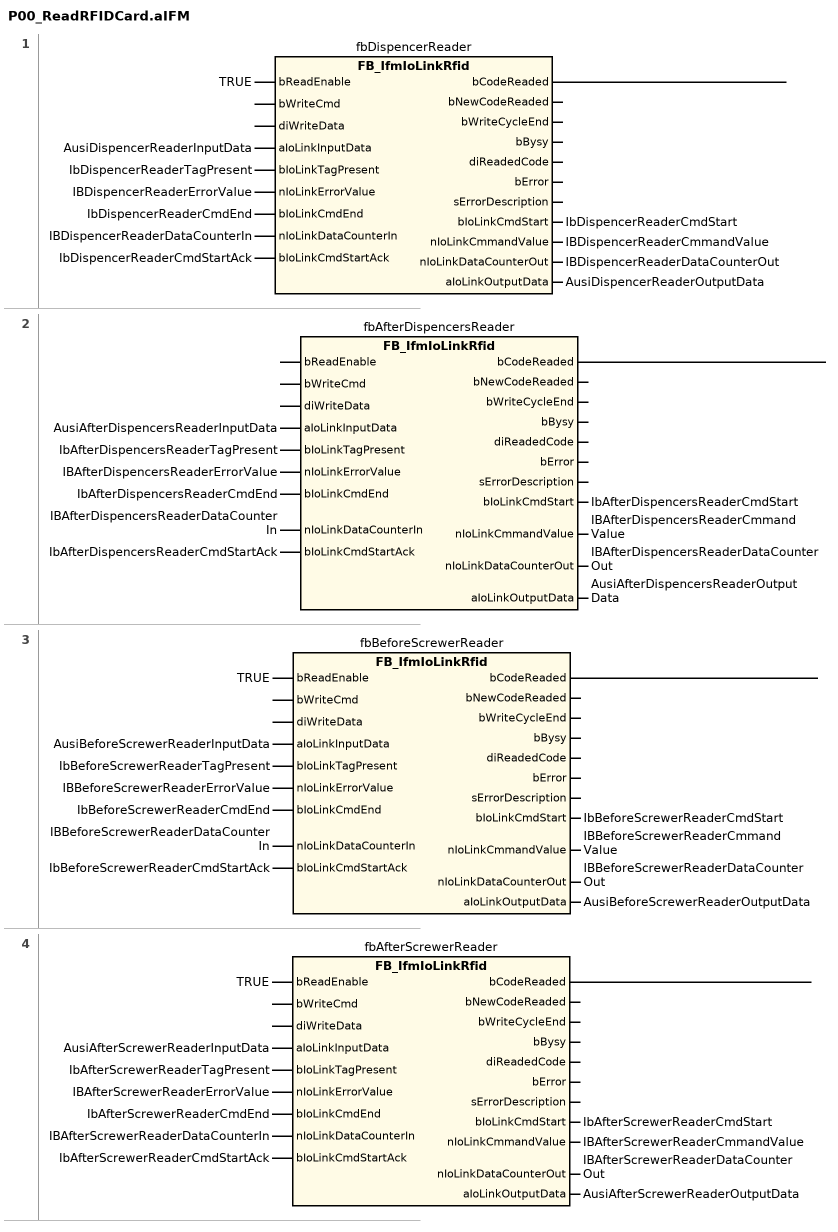
// NETWORK 1
fbDispencerReader(
    bReadEnable := TRUE,
    aIoLinkInputData := AusiDispencerReaderInputData,
    bIoLinkTagPresent := IbDispencerReaderTagPresent,
    nIoLinkErrorValue := IBDispencerReaderErrorValue,
    bIoLinkCmdEnd := IbDispencerReaderCmdEnd,
    nIoLinkDataCounterIn := IBDispencerReaderDataCounterIn,
    bIoLinkCmdStartAck := IbDispencerReaderCmdStartAck,
    bIoLinkCmdStart => IbDispencerReaderCmdStart,
    nIoLinkCmmandValue => IBDispencerReaderCmmandValue,
    nIoLinkDataCounterOut => IBDispencerReaderDataCounterOut,
    aIoLinkOutputData => AusiDispencerReaderOutputData); // FB_IfmIoLinkRfid

// NETWORK 2
fbAfterDispencersReader(
    aIoLinkInputData := AusiAfterDispencersReaderInputData,
    bIoLinkTagPresent := IbAfterDispencersReaderTagPresent,
    nIoLinkErrorValue := IBAfterDispencersReaderErrorValue,
    bIoLinkCmdEnd := IbAfterDispencersReaderCmdEnd,
    nIoLinkDataCounterIn := IBAfterDispencersReaderDataCounterIn,
    bIoLinkCmdStartAck := IbAfterDispencersReaderCmdStartAck,
    bIoLinkCmdStart => IbAfterDispencersReaderCmdStart,
    nIoLinkCmmandValue => IBAfterDispencersReaderCmmandValue,
    nIoLinkDataCounterOut => IBAfterDispencersReaderDataCounterOut,
    aIoLinkOutputData => AusiAfterDispencersReaderOutputData); // FB_IfmIoLinkRfid

// NETWORK 3
fbBeforeScrewerReader(
    bReadEnable := TRUE,
    aIoLinkInputData := AusiBeforeScrewerReaderInputData,
    bIoLinkTagPresent := IbBeforeScrewerReaderTagPresent,
    nIoLinkErrorValue := IBBeforeScrewerReaderErrorValue,
    bIoLinkCmdEnd := IbBeforeScrewerReaderCmdEnd,
    nIoLinkDataCounterIn := IBBeforeScrewerReaderDataCounterIn,
    bIoLinkCmdStartAck := IbBeforeScrewerReaderCmdStartAck,
    bIoLinkCmdStart => IbBeforeScrewerReaderCmdStart,
    nIoLinkCmmandValue => IBBeforeScrewerReaderCmmandValue,
    nIoLinkDataCounterOut => IBBeforeScrewerReaderDataCounterOut,
    aIoLinkOutputData => AusiBeforeScrewerReaderOutputData); // FB_IfmIoLinkRfid

// NETWORK 4
fbAfterScrewerReader(
    bReadEnable := TRUE,
    aIoLinkInputData := AusiAfterScrewerReaderInputData,
    bIoLinkTagPresent := IbAfterScrewerReaderTagPresent,
    nIoLinkErrorValue := IBAfterScrewerReaderErrorValue,
    bIoLinkCmdEnd := IbAfterScrewerReaderCmdEnd,
    nIoLinkDataCounterIn := IBAfterScrewerReaderDataCounterIn,
    bIoLinkCmdStartAck := IbAfterScrewerReaderCmdStartAck,
    bIoLinkCmdStart => IbAfterScrewerReaderCmdStart,
    nIoLinkCmmandValue => IBAfterScrewerReaderCmmandValue,
    nIoLinkDataCounterOut => IBAfterScrewerReaderDataCounterOut,
    aIoLinkOutputData => AusiAfterScrewerReaderOutputData); // FB_IfmIoLinkRfid

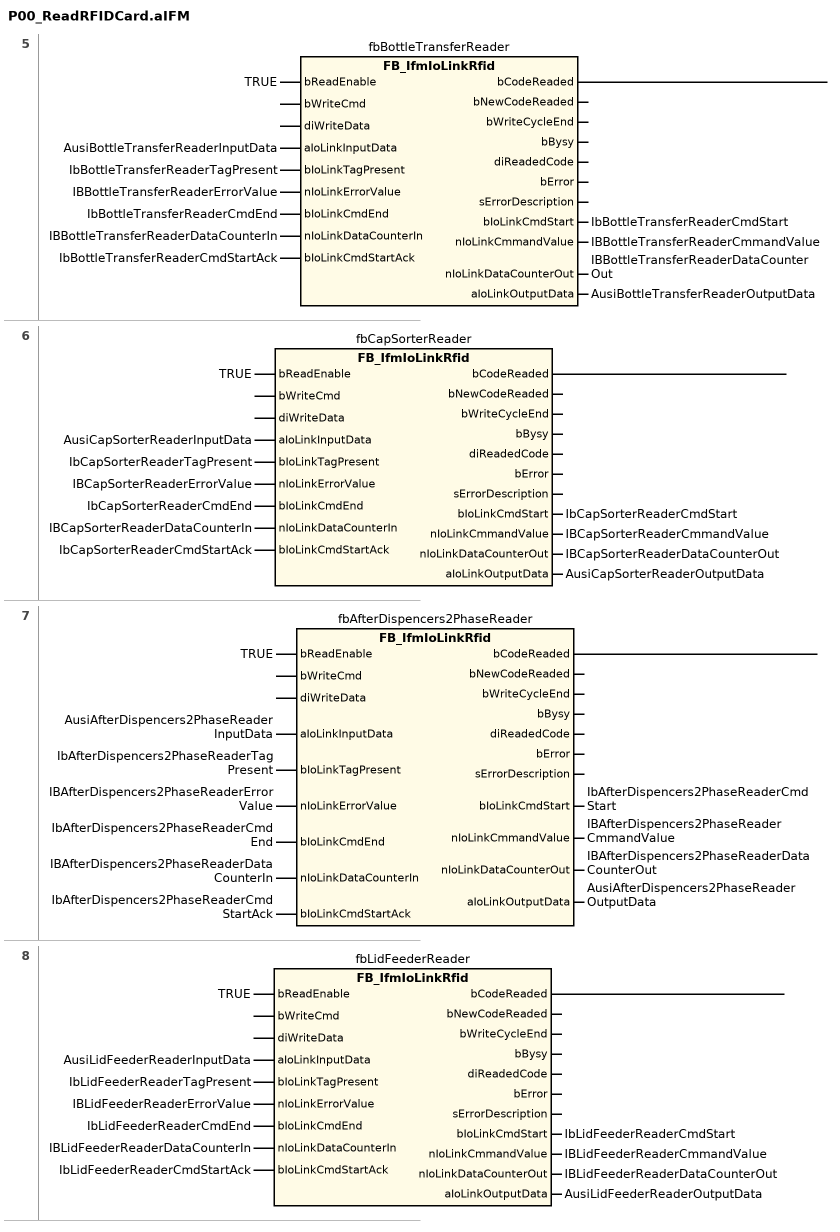
// NETWORK 5
fbBottleTransferReader(
    bReadEnable := TRUE,
    aIoLinkInputData := AusiBottleTransferReaderInputData,
    bIoLinkTagPresent := IbBottleTransferReaderTagPresent,
    nIoLinkErrorValue := IBBottleTransferReaderErrorValue,
    bIoLinkCmdEnd := IbBottleTransferReaderCmdEnd,
    nIoLinkDataCounterIn := IBBottleTransferReaderDataCounterIn,
    bIoLinkCmdStartAck := IbBottleTransferReaderCmdStartAck,
    bIoLinkCmdStart => IbBottleTransferReaderCmdStart,
    nIoLinkCmmandValue => IBBottleTransferReaderCmmandValue,
    nIoLinkDataCounterOut => IBBottleTransferReaderDataCounterOut,
    aIoLinkOutputData => AusiBottleTransferReaderOutputData); // FB_IfmIoLinkRfid

// NETWORK 6
fbCapSorterReader(
    bReadEnable := TRUE,
    aIoLinkInputData := AusiCapSorterReaderInputData,
    bIoLinkTagPresent := IbCapSorterReaderTagPresent,
    nIoLinkErrorValue := IBCapSorterReaderErrorValue,
    bIoLinkCmdEnd := IbCapSorterReaderCmdEnd,
    nIoLinkDataCounterIn := IBCapSorterReaderDataCounterIn,
    bIoLinkCmdStartAck := IbCapSorterReaderCmdStartAck,
    bIoLinkCmdStart => IbCapSorterReaderCmdStart,
    nIoLinkCmmandValue => IBCapSorterReaderCmmandValue,
    nIoLinkDataCounterOut => IBCapSorterReaderDataCounterOut,
    aIoLinkOutputData => AusiCapSorterReaderOutputData); // FB_IfmIoLinkRfid

// NETWORK 7
fbAfterDispencers2PhaseReader(
    bReadEnable := TRUE,
    aIoLinkInputData := AusiAfterDispencers2PhaseReaderInputData,
    bIoLinkTagPresent := IbAfterDispencers2PhaseReaderTagPresent,
    nIoLinkErrorValue := IBAfterDispencers2PhaseReaderErrorValue,
    bIoLinkCmdEnd := IbAfterDispencers2PhaseReaderCmdEnd,
    nIoLinkDataCounterIn := IBAfterDispencers2PhaseReaderDataCounterIn,
    bIoLinkCmdStartAck := IbAfterDispencers2PhaseReaderCmdStartAck,
    bIoLinkCmdStart => IbAfterDispencers2PhaseReaderCmdStart,
    nIoLinkCmmandValue => IBAfterDispencers2PhaseReaderCmmandValue,
    nIoLinkDataCounterOut => IBAfterDispencers2PhaseReaderDataCounterOut,
    aIoLinkOutputData => AusiAfterDispencers2PhaseReaderOutputData); // FB_IfmIoLinkRfid

// NETWORK 8
fbLidFeederReader(
    bReadEnable := TRUE,
    aIoLinkInputData := AusiLidFeederReaderInputData,
    bIoLinkTagPresent := IbLidFeederReaderTagPresent,
    nIoLinkErrorValue := IBLidFeederReaderErrorValue,
    bIoLinkCmdEnd := IbLidFeederReaderCmdEnd,
    nIoLinkDataCounterIn := IBLidFeederReaderDataCounterIn,
    bIoLinkCmdStartAck := IbLidFeederReaderCmdStartAck,
    bIoLinkCmdStart => IbLidFeederReaderCmdStart,
    nIoLinkCmmandValue => IBLidFeederReaderCmmandValue,
    nIoLinkDataCounterOut => IBLidFeederReaderDataCounterOut,
    aIoLinkOutputData => AusiLidFeederReaderOutputData); // FB_IfmIoLinkRfid

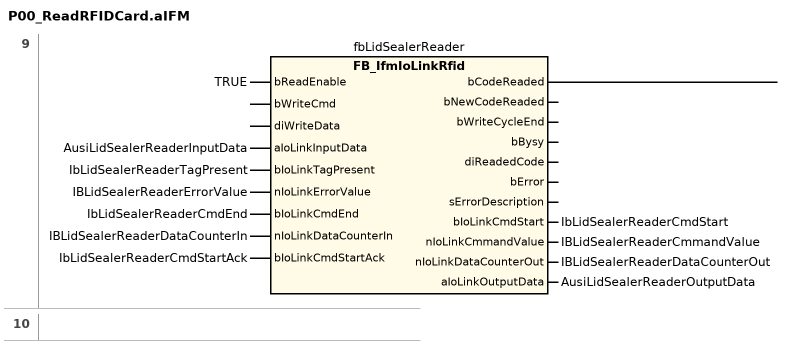
// NETWORK 9
fbLidSealerReader(
    bReadEnable := TRUE,
    aIoLinkInputData := AusiLidSealerReaderInputData,
    bIoLinkTagPresent := IbLidSealerReaderTagPresent,
    nIoLinkErrorValue := IBLidSealerReaderErrorValue,
    bIoLinkCmdEnd := IbLidSealerReaderCmdEnd,
    nIoLinkDataCounterIn := IBLidSealerReaderDataCounterIn,
    bIoLinkCmdStartAck := IbLidSealerReaderCmdStartAck,
    bIoLinkCmdStart => IbLidSealerReaderCmdStart,
    nIoLinkCmmandValue => IBLidSealerReaderCmmandValue,
    nIoLinkDataCounterOut => IBLidSealerReaderDataCounterOut,
    aIoLinkOutputData => AusiLidSealerReaderOutputData); // FB_IfmIoLinkRfid

// NETWORK 10
END_ACTION

ACTION aRFIDCheck:

//AnRFIDCardNumberShow							:ARRAY [1..100] OF ULINT;	// [H] Tabela numerów formatek 
IF VIS.AnRFIDWeightShow[1] = 0 THEN
	bRFIDCheckEnable :=	FALSE;
END_IF
rtbWeighingFormDone								(CLK:=	MAIN.bWeighingFormDone OR (NOT bFirstCycle AND VIS.AnRFIDWeightShow[1] > 0), Q=>);
IF rtbWeighingFormDone.Q THEN
	bRFIDCheckEnable :=	TRUE;
END_IF


IF bRFIDCheckResetAll THEN
	FOR i := 1 TO 100 DO												// Krok 1 - Przepisanie numerów RFID po przeważaniu
			AStRFIDCheck[i].iNumber				:=	0;
			AStRFIDCheck[i].iReaded1			:=	0;
			AStRFIDCheck[i].iReaded2			:=	0;
			AStRFIDCheck[i].iReaded3			:=	0;
			AStRFIDCheck[i].iReaded4			:=	0;
			AStRFIDCheck[i].iReaded5			:=	0;
	END_FOR		
	bRFIDCheckResetAll	:= FALSE;
END_IF

IF bRFIDCheckReset THEN
	FOR i := 1 TO 100 DO												// Krok 1 - Przepisanie numerów RFID po przeważaniu
			AStRFIDCheck[i].iReaded1			:=	0;
			AStRFIDCheck[i].iReaded2			:=	0;
			AStRFIDCheck[i].iReaded3			:=	0;
			AStRFIDCheck[i].iReaded4			:=	0;
			AStRFIDCheck[i].iReaded5			:=	0;
	END_FOR	
	
	iRFIDCheckNumberOfFormsExecute 			:= 0;
	iRFIDCheckProblemWithNumber				:= 0;
	iRFIDCheckDispencerWarning				:= 0;
	iRFIDCheckWeightWarning					:= 0;		
	iRFIDCheckBeforeScrewerWarning			:= 0;	
	iRFIDCheckAfterScrewerWarning			:= 0;	
	iRFIDCheckBottleTransferWarning			:= 0;		
	iRFIDReaded1Errors						:= 0;
	iRFIDReaded2Errors						:= 0;
	iRFIDReaded3Errors						:= 0;
	iRFIDReaded4Errors						:= 0;
	iRFIDReaded5Errors						:= 0;
	bRFIDCheckReset	:= FALSE;
END_IF


//Kasowanie w trakcie pracy i jak jest git

tonRFIDReset
	(IN:= P00_PackML.fbPMLAuto.ePMLState = Tc3_PackML.E_PMLState.ePMLState_EXECUTE AND
	iRFIDCheckDispencerWarning = iRFIDCheckDispencerWarningLast AND
	iRFIDCheckWeightWarning = iRFIDCheckWeightWarningLast AND
	iRFIDCheckBeforeScrewerWarning = iRFIDCheckBeforeScrewerWarningLast AND
	iRFIDCheckAfterScrewerWarning = iRFIDCheckAfterScrewerWarningLast AND
	iRFIDCheckBottleTransferWarning = iRFIDCheckBottleTransferWarningLast AND
	
	NOT tonRFIDReset.Q
	,PT := T#3M);

//Zapamietywanie ilości formatek po przewazaniu
IF rtbWeighingFormDone.Q OR bCycleReseting THEN	
	iRFIDCheckNumberOfFormsExecute 			:= 0;
	iRFIDCheckNumberOfFormsAfterWeighting 	:= 0;
	iRFIDCheckProblemWithNumber				:= 0;
	sRFIDInfoSensorError					:= '';
	iRFIDCheckDispencerWarning				:= 0;
	iRFIDCheckWeightWarning					:= 0;		
	iRFIDCheckBeforeScrewerWarning			:= 0;	
	iRFIDCheckAfterScrewerWarning			:= 0;	
	iRFIDCheckBottleTransferWarning			:= 0;	
	FOR i := 1 TO 100 DO												// Krok 1 - Przepisanie numerów RFID po przeważaniu
		IF VIS.AnRFIDCardNumberShow[i] > 0 THEN
			AStRFIDCheck[i].iNumber					:=	ULINT_TO_INT(VIS.AnRFIDCardNumberShow[i]);
			AStRFIDCheck[i].iReaded1				:=	0;
			AStRFIDCheck[i].iReaded2				:=	0;
			AStRFIDCheck[i].iReaded3				:=	0;
			AStRFIDCheck[i].iReaded4				:=	0;
			AStRFIDCheck[i].iReaded5				:=	0;		
			iRFIDCheckNumberOfFormsAfterWeighting	:=	iRFIDCheckNumberOfFormsAfterWeighting	+	1;
		END_IF
	END_FOR
END_IF

(*******************Reader1********************)
P00_ReadRFIDCard.bReadedCardDispencer;	nReadedCardDispencer;
tonRFIDCheckReader1Add	(IN:=	P00_ReadRFIDCard.bReadedCardDispencer,			PT:=T#10MS);
rtRFIDCheckReader1Add 	(CLK:=	tonRFIDCheckReader1Add.Q,						Q=>);
IF rtRFIDCheckReader1Add.Q AND bRFIDCheckEnable THEN
	FOR i:=1 TO 100 DO
		IF AStRFIDCheck[i].iNumber = ULINT_TO_INT(nReadedCardDispencer) THEN		// Krok 2 - Jeżei odczytało jakiś numer to dodaje +1
			AStRFIDCheck[i].iReaded1 := AStRFIDCheck[i].iReaded1	+	1;
			IF AStRFIDCheck[i].iReaded1 < -1 THEN AStRFIDCheck[i].iReaded1 := 0; END_IF // Jeżeli spowrotem odczytało to zeruj po jakims czasie
			IF AStRFIDCheck[i].iReaded1 > 1 THEN						// Krok 3 - Jeżei odczytało jakiś numer drugi raz to odejmuje od wszystkich -1
				FOR j:=1 TO 100 DO
					IF AStRFIDCheck[j].iNumber > 0 THEN
						AStRFIDCheck[j].iReaded1 := AStRFIDCheck[j].iReaded1	-	1;
					ELSE
						AStRFIDCheck[j].iReaded1 := 0;
					END_IF
				END_FOR				
			END_IF
			EXIT;
		END_IF	
	END_FOR
END_IF
(************Koniec Reader1*******************)

(*******************Reader2********************)
P00_ReadRFIDCard.bReadedCardAfterDispencers;	nReadedCardAfterDispencers;
tonRFIDCheckReader2Add	(IN:=	P00_ReadRFIDCard.bReadedCardAfterDispencers,	PT:=T#10MS);
rtRFIDCheckReader2Add 	(CLK:=	tonRFIDCheckReader2Add.Q,						Q=>);
IF rtRFIDCheckReader2Add.Q AND bRFIDCheckEnable THEN
	FOR i:=1 TO 100 DO
		IF AStRFIDCheck[i].iNumber = ULINT_TO_INT(nReadedCardAfterDispencers) THEN		// Krok 2 - Jeżei odczytało jakiś numer to dodaje +1
			AStRFIDCheck[i].iReaded2 := AStRFIDCheck[i].iReaded2	+	1;
			IF AStRFIDCheck[i].iReaded2 < -1 THEN AStRFIDCheck[i].iReaded2 := 0; END_IF // Jeżeli spowrotem odczytało to zeruj po jakims czasie
			IF AStRFIDCheck[i].iReaded2 > 1 THEN						// Krok 3 - Jeżei odczytało jakiś numer drugi raz to odejmuje od wszystkich -1
				FOR j:=1 TO 100 DO
					IF AStRFIDCheck[j].iNumber > 0 THEN
						AStRFIDCheck[j].iReaded2 := AStRFIDCheck[j].iReaded2	-	1;
					ELSE
						AStRFIDCheck[j].iReaded2 := 0;
					END_IF
				END_FOR				
			END_IF
			EXIT;
		END_IF	
	END_FOR
END_IF
(************Koniec Reader2*******************)

(*******************Reader3********************)
P00_ReadRFIDCard.bReadedCardBeforeScrewer;	nReadedCardBeforeScrewer;
tonRFIDCheckReader3Add	(IN:=	P00_ReadRFIDCard.bReadedCardBeforeScrewer,		PT:=T#10MS);
rtRFIDCheckReader3Add 	(CLK:=	tonRFIDCheckReader3Add.Q,						Q=>);
IF rtRFIDCheckReader3Add.Q AND bRFIDCheckEnable THEN
	FOR i:=1 TO 100 DO
		IF AStRFIDCheck[i].iNumber = ULINT_TO_INT(nReadedCardBeforeScrewer) THEN		// Krok 2 - Jeżei odczytało jakiś numer to dodaje +1
			AStRFIDCheck[i].iReaded3 := AStRFIDCheck[i].iReaded3	+	1;
			IF AStRFIDCheck[i].iReaded3 < -1 THEN AStRFIDCheck[i].iReaded3 := 0; END_IF // Jeżeli spowrotem odczytało to zeruj po jakims czasie			
			IF AStRFIDCheck[i].iReaded3 > 1 THEN						// Krok 3 - Jeżei odczytało jakiś numer drugi raz to odejmuje od wszystkich -1
				FOR j:=1 TO 100 DO
					IF AStRFIDCheck[j].iNumber > 0 THEN
						AStRFIDCheck[j].iReaded3 := AStRFIDCheck[j].iReaded3	-	1;
					ELSE
						AStRFIDCheck[j].iReaded3 := 0;
					END_IF
				END_FOR				
			END_IF
			EXIT;
		END_IF	
	END_FOR
END_IF
(************Koniec Reader3*******************)

(*******************Reader4********************)
P00_ReadRFIDCard.bReadedCardAfterScrewer;	nReadedCardAfterScrewer;
tonRFIDCheckReader4Add	(IN:=	P00_ReadRFIDCard.bReadedCardAfterScrewer,		PT:=T#10MS);
rtRFIDCheckReader4Add 	(CLK:=	tonRFIDCheckReader4Add.Q,						Q=>);
IF rtRFIDCheckReader4Add.Q AND bRFIDCheckEnable THEN
	FOR i:=1 TO 100 DO
		IF AStRFIDCheck[i].iNumber = ULINT_TO_INT(nReadedCardAfterScrewer) THEN		// Krok 2 - Jeżei odczytało jakiś numer to dodaje +1
			AStRFIDCheck[i].iReaded4 := AStRFIDCheck[i].iReaded4	+	1;
			IF AStRFIDCheck[i].iReaded4 < -1 THEN AStRFIDCheck[i].iReaded4 := 0; END_IF // Jeżeli spowrotem odczytało to zeruj po jakims czasie			
			IF AStRFIDCheck[i].iReaded4 > 1 THEN						// Krok 3 - Jeżei odczytało jakiś numer drugi raz to odejmuje od wszystkich -1
				FOR j:=1 TO 100 DO
					IF AStRFIDCheck[j].iNumber > 0 THEN
						AStRFIDCheck[j].iReaded4 := AStRFIDCheck[j].iReaded4	-	1;
					ELSE
						AStRFIDCheck[j].iReaded4 := 0;
					END_IF
				END_FOR				
			END_IF
			EXIT;
		END_IF	
	END_FOR
END_IF
(************Koniec Reader4*******************)

(*******************Reader5********************)
P00_ReadRFIDCard.bReadedCardBottleTransfer;	nReadedCardBottleTransfer;
tonRFIDCheckReader5Add	(IN:=	P00_ReadRFIDCard.bReadedCardBottleTransfer,		PT:=T#10MS);
rtRFIDCheckReader5Add 	(CLK:=	tonRFIDCheckReader5Add.Q,						Q=>);
IF rtRFIDCheckReader5Add.Q AND bRFIDCheckEnable THEN
	FOR i:=1 TO 100 DO
		IF AStRFIDCheck[i].iNumber = ULINT_TO_INT(nReadedCardBottleTransfer) THEN		// Krok 2 - Jeżei odczytało jakiś numer to dodaje +1
			AStRFIDCheck[i].iReaded5 := AStRFIDCheck[i].iReaded5	+	1;
			IF AStRFIDCheck[i].iReaded5 < -1 THEN AStRFIDCheck[i].iReaded5 := 0; END_IF // Jeżeli spowrotem odczytało to zeruj po jakims czasie			
			IF AStRFIDCheck[i].iReaded5 > 1 THEN						// Krok 3 - Jeżei odczytało jakiś numer drugi raz to odejmuje od wszystkich -1
				FOR j:=1 TO 100 DO
					IF AStRFIDCheck[j].iNumber > 0 THEN
						AStRFIDCheck[j].iReaded5 := AStRFIDCheck[j].iReaded5	-	1;
					ELSE
						AStRFIDCheck[j].iReaded5 := 0;
					END_IF
				END_FOR				
			END_IF
			EXIT;
		END_IF	
	END_FOR
END_IF
(************Koniec Reader5*******************)

//NoOfPucks:49/50;Error:13;Sensor:Dispencers
VIS.sSlowestStation4 := sRFIDInfo; 
sRFIDInfo := Concat(Concat(Concat(Concat(Concat('Pucks:',Concat(INT_TO_STRING(iRFIDCheckNumberOfFormsExecute),Concat('/',INT_TO_STRING(iRFIDCheckNumberOfFormsAfterWeighting)))),';FaultOrMiss:'),
									INT_TO_STRING(iRFIDCheckProblemWithNumber)),
									';SensorFault:'),
									sRFIDInfoSensorError)
;

tonRFIDCheck10s(IN:=NOT tonRFIDCheck10s.Q, PT:=T#15S);
IF tonRFIDCheck10s.Q AND bRFIDCheckEnable THEN
	iRFIDCheckNumberOfFormsExecute	:=	0;
	iRFIDReaded1Errors	:=	0;
	iRFIDReaded2Errors	:=	0;
	iRFIDReaded3Errors	:=	0;	
	iRFIDReaded4Errors	:=	0;	
	iRFIDReaded5Errors	:=	0;	
	FOR i:=1 TO 100 DO
			IF AStRFIDCheck[i].iNumber > 0 AND 									// Ilość formatek na lini
				(
					AStRFIDCheck[i].iReaded1 >=0 OR 		
					AStRFIDCheck[i].iReaded2 >=0 OR 					
					AStRFIDCheck[i].iReaded3 >=0 OR 	
					AStRFIDCheck[i].iReaded4 >=0 OR 	
					AStRFIDCheck[i].iReaded5 >=0  	
				)	
				AND
				NOT
				( 
					(AStRFIDCheck[i].iReaded1 < 0) AND 		
					(AStRFIDCheck[i].iReaded2 < 0) AND 					
					(AStRFIDCheck[i].iReaded3 < 0) AND  	
					(AStRFIDCheck[i].iReaded4 < 0) AND  	
					(AStRFIDCheck[i].iReaded5 < 0)  	
				)					
			THEN
				iRFIDCheckNumberOfFormsExecute	:=	iRFIDCheckNumberOfFormsExecute + 1;
			END_IF		
	END_FOR	
	FOR i:=1 TO 100 DO
			iRFIDCheckProblemWithNumber	:=	0;
			IF AStRFIDCheck[i].iNumber > 0 AND 									// Problem z tym numerem RFID
				(
					(AStRFIDCheck[i].iReaded1 < -3) OR		
					(AStRFIDCheck[i].iReaded2 < -3) OR					
					(AStRFIDCheck[i].iReaded3 < -3) OR 	
					(AStRFIDCheck[i].iReaded4 < -3) OR 	
					(AStRFIDCheck[i].iReaded5 < -3)  	
				)	
			THEN
				iRFIDCheckProblemWithNumber	:=	ULINT_TO_INT(AStRFIDCheck[i].iNumber);
				EXIT;
			END_IF		
	END_FOR	
	
	FOR i:=1 TO 100 DO
			sRFIDInfoSensorError	:=	'';

			IF AStRFIDCheck[i].iNumber > 0 AND AStRFIDCheck[i].iReaded1 < -3 THEN		iRFIDReaded1Errors	:=	iRFIDReaded1Errors	+	1;		END_IF	
			IF AStRFIDCheck[i].iNumber > 0 AND AStRFIDCheck[i].iReaded2 < -3 THEN		iRFIDReaded2Errors	:=	iRFIDReaded2Errors	+	1;		END_IF	
			IF AStRFIDCheck[i].iNumber > 0 AND AStRFIDCheck[i].iReaded3 < -3 THEN		iRFIDReaded3Errors	:=	iRFIDReaded3Errors	+	1;		END_IF	
			IF AStRFIDCheck[i].iNumber > 0 AND AStRFIDCheck[i].iReaded4 < -3 THEN		iRFIDReaded4Errors	:=	iRFIDReaded4Errors	+	1;		END_IF	
			IF AStRFIDCheck[i].iNumber > 0 AND AStRFIDCheck[i].iReaded5 < -3 THEN		iRFIDReaded5Errors	:=	iRFIDReaded5Errors	+	1;		END_IF	
				
	END_FOR		
				
	IF	iRFIDCheckDispencerWarning			>	2 OR
		iRFIDCheckWeightWarning				>	2 OR
		iRFIDCheckBeforeScrewerWarning		>	2 OR
		iRFIDCheckAfterScrewerWarning		>	2 OR
		iRFIDCheckBottleTransferWarning		>	2 			
	THEN
			
		IF		iRFIDCheckDispencerWarning			>	2 OR iRFIDReaded1Errors > 3 THEN	sRFIDInfoSensorError :=	'BeforeDispenser';
		ELSIF	iRFIDCheckWeightWarning				>	2 OR iRFIDReaded2Errors > 3 THEN	sRFIDInfoSensorError :=	'BeforeWeight';
		ELSIF	iRFIDCheckBeforeScrewerWarning		>	2 OR iRFIDReaded3Errors > 3 THEN	sRFIDInfoSensorError :=	'BeforeScrewer';
		ELSIF	iRFIDCheckAfterScrewerWarning		>	2 OR iRFIDReaded4Errors > 3 THEN	sRFIDInfoSensorError :=	'AfterScrewer';
		ELSIF	iRFIDCheckBottleTransferWarning		>	2 OR iRFIDReaded5Errors > 3 THEN	sRFIDInfoSensorError :=	'Robot';
		ELSE																				sRFIDInfoSensorError :=	'';
		END_IF						
			
	END_IF	
	
	IF iRFIDCheckProblemWithNumber = 0 THEN //kasowanie jak nie ma problemu z odczytem ??
		(*iRFIDCheckDispencerWarning	:=	0;	
		iRFIDCheckWeightWarning			:=	0;			
		iRFIDCheckBeforeScrewerWarning	:=	0;		
		iRFIDCheckAfterScrewerWarning	:=	0;			
		iRFIDCheckBottleTransferWarning	:=	0;*)		
	END_IF
	
	
END_IF

//Przykład
(*
5			1		1		1		1		1
2			1		0				1		1		
4			1		1		1		1		1
11
5
0
0

*)
AStRFIDCheck[1].iNumber;	AStRFIDCheck[1].iReaded1;		AStRFIDCheck[1].iReaded2;		AStRFIDCheck[1].iReaded3;		AStRFIDCheck[1].iReaded4;		AStRFIDCheck[1].iReaded5;
AStRFIDCheck[2].iNumber;	AStRFIDCheck[2].iReaded1;		AStRFIDCheck[2].iReaded2;		AStRFIDCheck[2].iReaded3;		AStRFIDCheck[2].iReaded4;		AStRFIDCheck[2].iReaded5;
AStRFIDCheck[3].iNumber;	AStRFIDCheck[3].iReaded1;		AStRFIDCheck[3].iReaded2;		AStRFIDCheck[3].iReaded3;		AStRFIDCheck[3].iReaded4;		AStRFIDCheck[3].iReaded5;
AStRFIDCheck[4].iNumber;	AStRFIDCheck[4].iReaded1;		AStRFIDCheck[4].iReaded2;		AStRFIDCheck[4].iReaded3;		AStRFIDCheck[4].iReaded4;		AStRFIDCheck[4].iReaded5;
AStRFIDCheck[5].iNumber;	AStRFIDCheck[5].iReaded1;		AStRFIDCheck[5].iReaded2;		AStRFIDCheck[5].iReaded3;		AStRFIDCheck[5].iReaded4;		AStRFIDCheck[5].iReaded5;
AStRFIDCheck[6].iNumber;	AStRFIDCheck[6].iReaded1;		AStRFIDCheck[6].iReaded2;		AStRFIDCheck[6].iReaded3;		AStRFIDCheck[6].iReaded4;		AStRFIDCheck[6].iReaded5;
AStRFIDCheck[7].iNumber;	AStRFIDCheck[7].iReaded1;		AStRFIDCheck[7].iReaded2;		AStRFIDCheck[7].iReaded3;		AStRFIDCheck[7].iReaded4;		AStRFIDCheck[7].iReaded5;
AStRFIDCheck[8].iNumber;	AStRFIDCheck[8].iReaded1;		AStRFIDCheck[8].iReaded2;		AStRFIDCheck[8].iReaded3;		AStRFIDCheck[8].iReaded4;		AStRFIDCheck[8].iReaded5;
AStRFIDCheck[9].iNumber;	AStRFIDCheck[9].iReaded1;		AStRFIDCheck[9].iReaded2;		AStRFIDCheck[9].iReaded3;		AStRFIDCheck[9].iReaded4;		AStRFIDCheck[9].iReaded5;
AStRFIDCheck[10].iNumber;	AStRFIDCheck[10].iReaded1;	AStRFIDCheck[10].iReaded2;	AStRFIDCheck[10].iReaded3;	AStRFIDCheck[10].iReaded4;	AStRFIDCheck[10].iReaded5;
AStRFIDCheck[11].iNumber;	AStRFIDCheck[11].iReaded1;	AStRFIDCheck[11].iReaded2;	AStRFIDCheck[11].iReaded3;	AStRFIDCheck[11].iReaded4;	AStRFIDCheck[11].iReaded5;
AStRFIDCheck[12].iNumber;	AStRFIDCheck[12].iReaded1;	AStRFIDCheck[12].iReaded2;	AStRFIDCheck[12].iReaded3;	AStRFIDCheck[12].iReaded4;	AStRFIDCheck[12].iReaded5;
AStRFIDCheck[13].iNumber;	AStRFIDCheck[13].iReaded1;	AStRFIDCheck[13].iReaded2;	AStRFIDCheck[13].iReaded3;	AStRFIDCheck[13].iReaded4;	AStRFIDCheck[13].iReaded5;
AStRFIDCheck[14].iNumber;	AStRFIDCheck[14].iReaded1;	AStRFIDCheck[14].iReaded2;	AStRFIDCheck[14].iReaded3;	AStRFIDCheck[14].iReaded4;	AStRFIDCheck[14].iReaded5;
AStRFIDCheck[15].iNumber;	AStRFIDCheck[15].iReaded1;	AStRFIDCheck[15].iReaded2;	AStRFIDCheck[15].iReaded3;	AStRFIDCheck[15].iReaded4;	AStRFIDCheck[15].iReaded5;
AStRFIDCheck[16].iNumber;	AStRFIDCheck[16].iReaded1;	AStRFIDCheck[16].iReaded2;	AStRFIDCheck[16].iReaded3;	AStRFIDCheck[16].iReaded4;	AStRFIDCheck[16].iReaded5;
AStRFIDCheck[17].iNumber;	AStRFIDCheck[17].iReaded1;	AStRFIDCheck[17].iReaded2;	AStRFIDCheck[17].iReaded3;	AStRFIDCheck[17].iReaded4;	AStRFIDCheck[17].iReaded5;
AStRFIDCheck[18].iNumber;	AStRFIDCheck[18].iReaded1;	AStRFIDCheck[18].iReaded2;	AStRFIDCheck[18].iReaded3;	AStRFIDCheck[18].iReaded4;	AStRFIDCheck[18].iReaded5;
AStRFIDCheck[19].iNumber;	AStRFIDCheck[19].iReaded1;	AStRFIDCheck[19].iReaded2;	AStRFIDCheck[19].iReaded3;	AStRFIDCheck[19].iReaded4;	AStRFIDCheck[19].iReaded5;
AStRFIDCheck[20].iNumber;	AStRFIDCheck[20].iReaded1;	AStRFIDCheck[20].iReaded2;	AStRFIDCheck[20].iReaded3;	AStRFIDCheck[20].iReaded4;	AStRFIDCheck[20].iReaded5;
AStRFIDCheck[21].iNumber;	AStRFIDCheck[21].iReaded1;	AStRFIDCheck[21].iReaded2;	AStRFIDCheck[21].iReaded3;	AStRFIDCheck[21].iReaded4;	AStRFIDCheck[21].iReaded5;
AStRFIDCheck[22].iNumber;	AStRFIDCheck[22].iReaded1;	AStRFIDCheck[22].iReaded2;	AStRFIDCheck[22].iReaded3;	AStRFIDCheck[22].iReaded4;	AStRFIDCheck[22].iReaded5;
AStRFIDCheck[23].iNumber;	AStRFIDCheck[23].iReaded1;	AStRFIDCheck[23].iReaded2;	AStRFIDCheck[23].iReaded3;	AStRFIDCheck[23].iReaded4;	AStRFIDCheck[23].iReaded5;
AStRFIDCheck[24].iNumber;	AStRFIDCheck[24].iReaded1;	AStRFIDCheck[24].iReaded2;	AStRFIDCheck[24].iReaded3;	AStRFIDCheck[24].iReaded4;	AStRFIDCheck[24].iReaded5;
AStRFIDCheck[25].iNumber;	AStRFIDCheck[25].iReaded1;	AStRFIDCheck[25].iReaded2;	AStRFIDCheck[25].iReaded3;	AStRFIDCheck[25].iReaded4;	AStRFIDCheck[25].iReaded5;
AStRFIDCheck[26].iNumber;	AStRFIDCheck[26].iReaded1;	AStRFIDCheck[26].iReaded2;	AStRFIDCheck[26].iReaded3;	AStRFIDCheck[26].iReaded4;	AStRFIDCheck[26].iReaded5;
AStRFIDCheck[27].iNumber;	AStRFIDCheck[27].iReaded1;	AStRFIDCheck[27].iReaded2;	AStRFIDCheck[27].iReaded3;	AStRFIDCheck[27].iReaded4;	AStRFIDCheck[27].iReaded5;
AStRFIDCheck[28].iNumber;	AStRFIDCheck[28].iReaded1;	AStRFIDCheck[28].iReaded2;	AStRFIDCheck[28].iReaded3;	AStRFIDCheck[28].iReaded4;	AStRFIDCheck[28].iReaded5;
AStRFIDCheck[29].iNumber;	AStRFIDCheck[29].iReaded1;	AStRFIDCheck[29].iReaded2;	AStRFIDCheck[29].iReaded3;	AStRFIDCheck[29].iReaded4;	AStRFIDCheck[29].iReaded5;
AStRFIDCheck[30].iNumber;	AStRFIDCheck[30].iReaded1;	AStRFIDCheck[30].iReaded2;	AStRFIDCheck[30].iReaded3;	AStRFIDCheck[30].iReaded4;	AStRFIDCheck[30].iReaded5;
AStRFIDCheck[31].iNumber;	AStRFIDCheck[31].iReaded1;	AStRFIDCheck[31].iReaded2;	AStRFIDCheck[31].iReaded3;	AStRFIDCheck[31].iReaded4;	AStRFIDCheck[31].iReaded5;
AStRFIDCheck[32].iNumber;	AStRFIDCheck[32].iReaded1;	AStRFIDCheck[32].iReaded2;	AStRFIDCheck[32].iReaded3;	AStRFIDCheck[32].iReaded4;	AStRFIDCheck[32].iReaded5;
AStRFIDCheck[33].iNumber;	AStRFIDCheck[33].iReaded1;	AStRFIDCheck[33].iReaded2;	AStRFIDCheck[33].iReaded3;	AStRFIDCheck[33].iReaded4;	AStRFIDCheck[33].iReaded5;
AStRFIDCheck[34].iNumber;	AStRFIDCheck[34].iReaded1;	AStRFIDCheck[34].iReaded2;	AStRFIDCheck[34].iReaded3;	AStRFIDCheck[34].iReaded4;	AStRFIDCheck[34].iReaded5;
AStRFIDCheck[35].iNumber;	AStRFIDCheck[35].iReaded1;	AStRFIDCheck[35].iReaded2;	AStRFIDCheck[35].iReaded3;	AStRFIDCheck[35].iReaded4;	AStRFIDCheck[35].iReaded5;
AStRFIDCheck[36].iNumber;	AStRFIDCheck[36].iReaded1;	AStRFIDCheck[36].iReaded2;	AStRFIDCheck[36].iReaded3;	AStRFIDCheck[36].iReaded4;	AStRFIDCheck[36].iReaded5;
AStRFIDCheck[37].iNumber;	AStRFIDCheck[37].iReaded1;	AStRFIDCheck[37].iReaded2;	AStRFIDCheck[37].iReaded3;	AStRFIDCheck[37].iReaded4;	AStRFIDCheck[37].iReaded5;
AStRFIDCheck[38].iNumber;	AStRFIDCheck[38].iReaded1;	AStRFIDCheck[38].iReaded2;	AStRFIDCheck[38].iReaded3;	AStRFIDCheck[38].iReaded4;	AStRFIDCheck[38].iReaded5;
AStRFIDCheck[39].iNumber;	AStRFIDCheck[39].iReaded1;	AStRFIDCheck[39].iReaded2;	AStRFIDCheck[39].iReaded3;	AStRFIDCheck[39].iReaded4;	AStRFIDCheck[39].iReaded5;
AStRFIDCheck[40].iNumber;	AStRFIDCheck[40].iReaded1;	AStRFIDCheck[40].iReaded2;	AStRFIDCheck[40].iReaded3;	AStRFIDCheck[40].iReaded4;	AStRFIDCheck[40].iReaded5;
AStRFIDCheck[41].iNumber;	AStRFIDCheck[41].iReaded1;	AStRFIDCheck[41].iReaded2;	AStRFIDCheck[41].iReaded3;	AStRFIDCheck[41].iReaded4;	AStRFIDCheck[41].iReaded5;
AStRFIDCheck[42].iNumber;	AStRFIDCheck[42].iReaded1;	AStRFIDCheck[42].iReaded2;	AStRFIDCheck[42].iReaded3;	AStRFIDCheck[42].iReaded4;	AStRFIDCheck[42].iReaded5;
AStRFIDCheck[43].iNumber;	AStRFIDCheck[43].iReaded1;	AStRFIDCheck[43].iReaded2;	AStRFIDCheck[43].iReaded3;	AStRFIDCheck[43].iReaded4;	AStRFIDCheck[43].iReaded5;
AStRFIDCheck[44].iNumber;	AStRFIDCheck[44].iReaded1;	AStRFIDCheck[44].iReaded2;	AStRFIDCheck[44].iReaded3;	AStRFIDCheck[44].iReaded4;	AStRFIDCheck[44].iReaded5;
AStRFIDCheck[45].iNumber;	AStRFIDCheck[45].iReaded1;	AStRFIDCheck[45].iReaded2;	AStRFIDCheck[45].iReaded3;	AStRFIDCheck[45].iReaded4;	AStRFIDCheck[45].iReaded5;
AStRFIDCheck[46].iNumber;	AStRFIDCheck[46].iReaded1;	AStRFIDCheck[46].iReaded2;	AStRFIDCheck[46].iReaded3;	AStRFIDCheck[46].iReaded4;	AStRFIDCheck[46].iReaded5;
AStRFIDCheck[47].iNumber;	AStRFIDCheck[47].iReaded1;	AStRFIDCheck[47].iReaded2;	AStRFIDCheck[47].iReaded3;	AStRFIDCheck[47].iReaded4;	AStRFIDCheck[47].iReaded5;
AStRFIDCheck[48].iNumber;	AStRFIDCheck[48].iReaded1;	AStRFIDCheck[48].iReaded2;	AStRFIDCheck[48].iReaded3;	AStRFIDCheck[48].iReaded4;	AStRFIDCheck[48].iReaded5;
AStRFIDCheck[49].iNumber;	AStRFIDCheck[49].iReaded1;	AStRFIDCheck[49].iReaded2;	AStRFIDCheck[49].iReaded3;	AStRFIDCheck[49].iReaded4;	AStRFIDCheck[49].iReaded5;
AStRFIDCheck[50].iNumber;	AStRFIDCheck[50].iReaded1;	AStRFIDCheck[50].iReaded2;	AStRFIDCheck[50].iReaded3;	AStRFIDCheck[50].iReaded4;	AStRFIDCheck[50].iReaded5;
AStRFIDCheck[51].iNumber;	AStRFIDCheck[51].iReaded1;	AStRFIDCheck[51].iReaded2;	AStRFIDCheck[51].iReaded3;	AStRFIDCheck[51].iReaded4;	AStRFIDCheck[51].iReaded5;
AStRFIDCheck[52].iNumber;	AStRFIDCheck[52].iReaded1;	AStRFIDCheck[52].iReaded2;	AStRFIDCheck[52].iReaded3;	AStRFIDCheck[52].iReaded4;	AStRFIDCheck[52].iReaded5;
AStRFIDCheck[53].iNumber;	AStRFIDCheck[53].iReaded1;	AStRFIDCheck[53].iReaded2;	AStRFIDCheck[53].iReaded3;	AStRFIDCheck[53].iReaded4;	AStRFIDCheck[53].iReaded5;
AStRFIDCheck[54].iNumber;	AStRFIDCheck[54].iReaded1;	AStRFIDCheck[54].iReaded2;	AStRFIDCheck[54].iReaded3;	AStRFIDCheck[54].iReaded4;	AStRFIDCheck[54].iReaded5;
AStRFIDCheck[55].iNumber;	AStRFIDCheck[55].iReaded1;	AStRFIDCheck[55].iReaded2;	AStRFIDCheck[55].iReaded3;	AStRFIDCheck[55].iReaded4;	AStRFIDCheck[55].iReaded5;
AStRFIDCheck[56].iNumber;	AStRFIDCheck[56].iReaded1;	AStRFIDCheck[56].iReaded2;	AStRFIDCheck[56].iReaded3;	AStRFIDCheck[56].iReaded4;	AStRFIDCheck[56].iReaded5;
AStRFIDCheck[57].iNumber;	AStRFIDCheck[57].iReaded1;	AStRFIDCheck[57].iReaded2;	AStRFIDCheck[57].iReaded3;	AStRFIDCheck[57].iReaded4;	AStRFIDCheck[57].iReaded5;
AStRFIDCheck[58].iNumber;	AStRFIDCheck[58].iReaded1;	AStRFIDCheck[58].iReaded2;	AStRFIDCheck[58].iReaded3;	AStRFIDCheck[58].iReaded4;	AStRFIDCheck[58].iReaded5;
AStRFIDCheck[59].iNumber;	AStRFIDCheck[59].iReaded1;	AStRFIDCheck[59].iReaded2;	AStRFIDCheck[59].iReaded3;	AStRFIDCheck[59].iReaded4;	AStRFIDCheck[59].iReaded5;
AStRFIDCheck[60].iNumber;	AStRFIDCheck[60].iReaded1;	AStRFIDCheck[60].iReaded2;	AStRFIDCheck[60].iReaded3;	AStRFIDCheck[60].iReaded4;	AStRFIDCheck[60].iReaded5;
AStRFIDCheck[61].iNumber;	AStRFIDCheck[61].iReaded1;	AStRFIDCheck[61].iReaded2;	AStRFIDCheck[61].iReaded3;	AStRFIDCheck[61].iReaded4;	AStRFIDCheck[61].iReaded5;
AStRFIDCheck[62].iNumber;	AStRFIDCheck[62].iReaded1;	AStRFIDCheck[62].iReaded2;	AStRFIDCheck[62].iReaded3;	AStRFIDCheck[62].iReaded4;	AStRFIDCheck[62].iReaded5;
AStRFIDCheck[63].iNumber;	AStRFIDCheck[63].iReaded1;	AStRFIDCheck[63].iReaded2;	AStRFIDCheck[63].iReaded3;	AStRFIDCheck[63].iReaded4;	AStRFIDCheck[63].iReaded5;
AStRFIDCheck[64].iNumber;	AStRFIDCheck[64].iReaded1;	AStRFIDCheck[64].iReaded2;	AStRFIDCheck[64].iReaded3;	AStRFIDCheck[64].iReaded4;	AStRFIDCheck[64].iReaded5;
AStRFIDCheck[65].iNumber;	AStRFIDCheck[65].iReaded1;	AStRFIDCheck[65].iReaded2;	AStRFIDCheck[65].iReaded3;	AStRFIDCheck[65].iReaded4;	AStRFIDCheck[65].iReaded5;
AStRFIDCheck[66].iNumber;	AStRFIDCheck[66].iReaded1;	AStRFIDCheck[66].iReaded2;	AStRFIDCheck[66].iReaded3;	AStRFIDCheck[66].iReaded4;	AStRFIDCheck[66].iReaded5;
AStRFIDCheck[67].iNumber;	AStRFIDCheck[67].iReaded1;	AStRFIDCheck[67].iReaded2;	AStRFIDCheck[67].iReaded3;	AStRFIDCheck[67].iReaded4;	AStRFIDCheck[67].iReaded5;
AStRFIDCheck[68].iNumber;	AStRFIDCheck[68].iReaded1;	AStRFIDCheck[68].iReaded2;	AStRFIDCheck[68].iReaded3;	AStRFIDCheck[68].iReaded4;	AStRFIDCheck[68].iReaded5;
AStRFIDCheck[69].iNumber;	AStRFIDCheck[69].iReaded1;	AStRFIDCheck[69].iReaded2;	AStRFIDCheck[69].iReaded3;	AStRFIDCheck[69].iReaded4;	AStRFIDCheck[69].iReaded5;
AStRFIDCheck[70].iNumber;	AStRFIDCheck[70].iReaded1;	AStRFIDCheck[70].iReaded2;	AStRFIDCheck[70].iReaded3;	AStRFIDCheck[70].iReaded4;	AStRFIDCheck[70].iReaded5;
AStRFIDCheck[71].iNumber;	AStRFIDCheck[71].iReaded1;	AStRFIDCheck[71].iReaded2;	AStRFIDCheck[71].iReaded3;	AStRFIDCheck[71].iReaded4;	AStRFIDCheck[71].iReaded5;
AStRFIDCheck[72].iNumber;	AStRFIDCheck[72].iReaded1;	AStRFIDCheck[72].iReaded2;	AStRFIDCheck[72].iReaded3;	AStRFIDCheck[72].iReaded4;	AStRFIDCheck[72].iReaded5;
AStRFIDCheck[73].iNumber;	AStRFIDCheck[73].iReaded1;	AStRFIDCheck[73].iReaded2;	AStRFIDCheck[73].iReaded3;	AStRFIDCheck[73].iReaded4;	AStRFIDCheck[73].iReaded5;
AStRFIDCheck[74].iNumber;	AStRFIDCheck[74].iReaded1;	AStRFIDCheck[74].iReaded2;	AStRFIDCheck[74].iReaded3;	AStRFIDCheck[74].iReaded4;	AStRFIDCheck[74].iReaded5;
AStRFIDCheck[75].iNumber;	AStRFIDCheck[75].iReaded1;	AStRFIDCheck[75].iReaded2;	AStRFIDCheck[75].iReaded3;	AStRFIDCheck[75].iReaded4;	AStRFIDCheck[75].iReaded5;
AStRFIDCheck[76].iNumber;	AStRFIDCheck[76].iReaded1;	AStRFIDCheck[76].iReaded2;	AStRFIDCheck[76].iReaded3;	AStRFIDCheck[76].iReaded4;	AStRFIDCheck[76].iReaded5;
AStRFIDCheck[77].iNumber;	AStRFIDCheck[77].iReaded1;	AStRFIDCheck[77].iReaded2;	AStRFIDCheck[77].iReaded3;	AStRFIDCheck[77].iReaded4;	AStRFIDCheck[77].iReaded5;
AStRFIDCheck[78].iNumber;	AStRFIDCheck[78].iReaded1;	AStRFIDCheck[78].iReaded2;	AStRFIDCheck[78].iReaded3;	AStRFIDCheck[78].iReaded4;	AStRFIDCheck[78].iReaded5;
AStRFIDCheck[79].iNumber;	AStRFIDCheck[79].iReaded1;	AStRFIDCheck[79].iReaded2;	AStRFIDCheck[79].iReaded3;	AStRFIDCheck[79].iReaded4;	AStRFIDCheck[79].iReaded5;
AStRFIDCheck[80].iNumber;	AStRFIDCheck[80].iReaded1;	AStRFIDCheck[80].iReaded2;	AStRFIDCheck[80].iReaded3;	AStRFIDCheck[80].iReaded4;	AStRFIDCheck[80].iReaded5;
AStRFIDCheck[81].iNumber;	AStRFIDCheck[81].iReaded1;	AStRFIDCheck[81].iReaded2;	AStRFIDCheck[81].iReaded3;	AStRFIDCheck[81].iReaded4;	AStRFIDCheck[81].iReaded5;
AStRFIDCheck[82].iNumber;	AStRFIDCheck[82].iReaded1;	AStRFIDCheck[82].iReaded2;	AStRFIDCheck[82].iReaded3;	AStRFIDCheck[82].iReaded4;	AStRFIDCheck[82].iReaded5;
AStRFIDCheck[83].iNumber;	AStRFIDCheck[83].iReaded1;	AStRFIDCheck[83].iReaded2;	AStRFIDCheck[83].iReaded3;	AStRFIDCheck[83].iReaded4;	AStRFIDCheck[83].iReaded5;
AStRFIDCheck[84].iNumber;	AStRFIDCheck[84].iReaded1;	AStRFIDCheck[84].iReaded2;	AStRFIDCheck[84].iReaded3;	AStRFIDCheck[84].iReaded4;	AStRFIDCheck[84].iReaded5;
AStRFIDCheck[85].iNumber;	AStRFIDCheck[85].iReaded1;	AStRFIDCheck[85].iReaded2;	AStRFIDCheck[85].iReaded3;	AStRFIDCheck[85].iReaded4;	AStRFIDCheck[85].iReaded5;
AStRFIDCheck[86].iNumber;	AStRFIDCheck[86].iReaded1;	AStRFIDCheck[86].iReaded2;	AStRFIDCheck[86].iReaded3;	AStRFIDCheck[86].iReaded4;	AStRFIDCheck[86].iReaded5;
AStRFIDCheck[87].iNumber;	AStRFIDCheck[87].iReaded1;	AStRFIDCheck[87].iReaded2;	AStRFIDCheck[87].iReaded3;	AStRFIDCheck[87].iReaded4;	AStRFIDCheck[87].iReaded5;
AStRFIDCheck[88].iNumber;	AStRFIDCheck[88].iReaded1;	AStRFIDCheck[88].iReaded2;	AStRFIDCheck[88].iReaded3;	AStRFIDCheck[88].iReaded4;	AStRFIDCheck[88].iReaded5;
AStRFIDCheck[89].iNumber;	AStRFIDCheck[89].iReaded1;	AStRFIDCheck[89].iReaded2;	AStRFIDCheck[89].iReaded3;	AStRFIDCheck[89].iReaded4;	AStRFIDCheck[89].iReaded5;
AStRFIDCheck[90].iNumber;	AStRFIDCheck[90].iReaded1;	AStRFIDCheck[90].iReaded2;	AStRFIDCheck[90].iReaded3;	AStRFIDCheck[90].iReaded4;	AStRFIDCheck[90].iReaded5;
AStRFIDCheck[91].iNumber;	AStRFIDCheck[91].iReaded1;	AStRFIDCheck[91].iReaded2;	AStRFIDCheck[91].iReaded3;	AStRFIDCheck[91].iReaded4;	AStRFIDCheck[91].iReaded5;
AStRFIDCheck[92].iNumber;	AStRFIDCheck[92].iReaded1;	AStRFIDCheck[92].iReaded2;	AStRFIDCheck[92].iReaded3;	AStRFIDCheck[92].iReaded4;	AStRFIDCheck[92].iReaded5;
AStRFIDCheck[93].iNumber;	AStRFIDCheck[93].iReaded1;	AStRFIDCheck[93].iReaded2;	AStRFIDCheck[93].iReaded3;	AStRFIDCheck[93].iReaded4;	AStRFIDCheck[93].iReaded5;
AStRFIDCheck[94].iNumber;	AStRFIDCheck[94].iReaded1;	AStRFIDCheck[94].iReaded2;	AStRFIDCheck[94].iReaded3;	AStRFIDCheck[94].iReaded4;	AStRFIDCheck[94].iReaded5;
AStRFIDCheck[95].iNumber;	AStRFIDCheck[95].iReaded1;	AStRFIDCheck[95].iReaded2;	AStRFIDCheck[95].iReaded3;	AStRFIDCheck[95].iReaded4;	AStRFIDCheck[95].iReaded5;
AStRFIDCheck[96].iNumber;	AStRFIDCheck[96].iReaded1;	AStRFIDCheck[96].iReaded2;	AStRFIDCheck[96].iReaded3;	AStRFIDCheck[96].iReaded4;	AStRFIDCheck[96].iReaded5;
AStRFIDCheck[97].iNumber;	AStRFIDCheck[97].iReaded1;	AStRFIDCheck[97].iReaded2;	AStRFIDCheck[97].iReaded3;	AStRFIDCheck[97].iReaded4;	AStRFIDCheck[97].iReaded5;
AStRFIDCheck[98].iNumber;	AStRFIDCheck[98].iReaded1;	AStRFIDCheck[98].iReaded2;	AStRFIDCheck[98].iReaded3;	AStRFIDCheck[98].iReaded4;	AStRFIDCheck[98].iReaded5;
AStRFIDCheck[99].iNumber;	AStRFIDCheck[99].iReaded1;	AStRFIDCheck[99].iReaded2;	AStRFIDCheck[99].iReaded3;	AStRFIDCheck[99].iReaded4;	AStRFIDCheck[99].iReaded5;
AStRFIDCheck[100].iNumber;	AStRFIDCheck[100].iReaded1;	AStRFIDCheck[100].iReaded2;	AStRFIDCheck[100].iReaded3;	AStRFIDCheck[100].iReaded4;	AStRFIDCheck[100].iReaded5;
END_ACTION

ACTION aRFIDCheck_1:



//	AnRFIDCardNumberShow							:ARRAY [1..100] OF ULINT;	// [H] Tabela numerów formatek 


(*rtbWeighingFormDone						(CLK:=MAIN.bWeighingFormDone, Q=>);
rtRFIDCheckbReadedCardBottleTransfer	(CLK:=P00_ReadRFIDCard.bReadedCardBottleTransfer AND P00_ReadRFIDCard.nReadedCardBottleTransfer > 0 AND 
										iRFIDCheck	=	30
										,Q=>);
IF rtRFIDCheckbReadedCardBottleTransfer.Q THEN
;
END_IF
//AnRFIDCardNumberShow							:ARRAY [1..100] OF ULINT;	// [H] Tabela numerów formatek 

//Zapamietywanie ilości formatek po przewazaniu
IF rtbWeighingFormDone.Q THEN
	iRFIDCheckNumberOfFormsExecute 			:= 0;
	iRFIDCheckNumberOfFormsAfterWeighting 	:= 0;
	sRFIDInfoSensorError					:= '';
	FOR i := 1 TO 100 DO
		IF VIS.AnRFIDCardNumberShow[i] > 0 THEN
			iRFIDCheckNumberOfFormsAfterWeighting :=	iRFIDCheckNumberOfFormsAfterWeighting	+	1;
		END_IF
	END_FOR
	
END_IF
//NoOfPucks:49/50;Error:13;Sensor:Dispencers
VIS.sSlowestStation4 := sRFIDInfo; {warning 'sSlowestStation5 usunąć używanie'}
sRFIDInfo := Concat(Concat(Concat(Concat(Concat('NoOfPucks:',Concat(INT_TO_STRING(iRFIDCheckNumberOfFormsExecute),Concat('/',INT_TO_STRING(iRFIDCheckNumberOfFormsAfterWeighting)))),';Error:'),
									INT_TO_STRING(iRFIDCheckProblemWithNumber)),
									';Sensor:'),
									sRFIDInfoSensorError)
;

//Jezeli start i wykryty jakiś numer
CASE iRFIDCheck OF
	0:
		iRFIDCheckDispencerWarning				:=	0;
		iRFIDCheckWeightWarning					:=	0;		
		iRFIDCheckBeforeScrewerWarning			:=	0;
		iRFIDCheckAfterScrewerWarning			:=	0;	
		iRFIDCheckBottleTransferWarning			:=	0;	
		iRFIDCheck	:=	iRFIDCheck	+	10;
		
	10: // 1 - Rozpoczaecie sprawdzania	
		IF 	P00_ReadRFIDCard.nReadedCardBottleTransfer > 0 AND 
			P00_ReadRFIDCard.nReadedCardBottleTransfer <> AuliRFIDCheck[1] AND 
			gvlUnit.eState = E_PackMLState.eExecute THEN
				iRFIDCheck	:=	iRFIDCheck	+	10;	
		END_IF
		
	20: // 2 - Wpisanie pierwszego wykrytego numeru i innego niż ostatni do tablicy RFID w cyklu	
		FOR i:=1 TO 100 DO
			AuliRFIDCheck[i]	:=	0;
		END_FOR
		iRFIDCheckNumberOfFormsExecuteTemp	:=	1;
		AuliRFIDCheck[1]					:=	P00_ReadRFIDCard.nReadedCardBottleTransfer;
		iRFIDCheck							:=	iRFIDCheck	+	10;	
		bRFIDCheckSave						:=	TRUE;
	30: // 3 - Tworzenie tablicy w cyklu
		AuliRFIDCheck[1];
		IF NOT (AuliRFIDCheck[1] = P00_ReadRFIDCard.nReadedCardBottleTransfer) THEN
				iRFIDTest	:=	iRFIDTest	+	1;
			IF rtRFIDCheckbReadedCardBottleTransfer.Q THEN //Jezeli nowy numer
				FOR i:=1 TO 100 DO //Czy jest już ten numer w tablicy?
					bRFIDCheckSave				:=	TRUE;
					IF	AuliRFIDCheck[i] = P00_ReadRFIDCard.nReadedCardBottleTransfer THEN
						bRFIDCheckSave			:=	FALSE;
						EXIT;
					END_IF
				END_FOR
			
				IF bRFIDCheckSave THEN //Dodaj nowy numer do tablicy
					iRFIDCheckNumberOfFormsExecuteTemp	:=	iRFIDCheckNumberOfFormsExecuteTemp	+	1;
					FOR i:=1 TO 100 DO
						IF AuliRFIDCheck[i] = 0 THEN
							AuliRFIDCheck[i]	:=	P00_ReadRFIDCard.nReadedCardBottleTransfer;
							EXIT;
						END_IF
					END_FOR
					bRFIDCheckSave				:=	FALSE;
				END_IF
			END_IF	
		ELSIF AuliRFIDCheck[1] = P00_ReadRFIDCard.nReadedCardBottleTransfer AND NOT bRFIDCheckSave THEN
			iRFIDCheck	:=	iRFIDCheck	+	10;	
		END_IF
			
		40: // 4 - Wykryto powtarzający się numer RFID wiec sprawdzanie czy jest to samo co w przeważaniu i zapisanie 1 numeru różniącego się
			FOR i:=1 TO 100 DO //Czy jest już ten numer w tablicy?
				FOR j:=1 TO 100 DO 
					bRFIDCheckDiffrence				:=	TRUE;				
					IF	AuliRFIDCheck[i] = VIS.AnRFIDCardNumberShow[j] THEN
						bRFIDCheckDiffrence				:=	FALSE;					
						EXIT;
					END_IF
				END_FOR			
				IF bRFIDCheckDiffrence THEN
					iRFIDCheckProblemWithNumber	:=	ULINT_TO_INT(AuliRFIDCheck[i]) ;
					EXIT;
				END_IF
			END_FOR		
			iRFIDCheck	:=	iRFIDCheck	+	10;	
			
		50: // 5 - Koniec sprawdzania, przepisanie wartości
			iRFIDCheckNumberOfFormsExecute	:=	iRFIDCheckNumberOfFormsExecuteTemp;
	
			IF		iRFIDCheckDispencerWarning			>	2 THEN	sRFIDInfoSensorError :=	'BeforeDispenser';
			ELSIF	iRFIDCheckWeightWarning				>	2 THEN	sRFIDInfoSensorError :=	'BeforeWeight';
			ELSIF	iRFIDCheckBeforeScrewerWarning		>	2 THEN	sRFIDInfoSensorError :=	'BeforeScrewer';
			ELSIF	iRFIDCheckAfterScrewerWarning		>	2 THEN	sRFIDInfoSensorError :=	'AfterScrewer';
			ELSIF	iRFIDCheckBottleTransferWarning		>	2 THEN	sRFIDInfoSensorError :=	'Robot';
			ELSE													sRFIDInfoSensorError :=	'';
			END_IF
			iRFIDCheck						:=	100;		
		60: 
			iRFIDCheck	:=	iRFIDCheck	+	10;		
		70: 
			iRFIDCheck	:=	iRFIDCheck	+	10;	
		80: 
			iRFIDCheck	:=	iRFIDCheck	+	10;		
		90: 
			iRFIDCheck	:=	iRFIDCheck	+	10;	
		100: 
			iRFIDCheck	:=	0;		
END_CASE


AuliRFIDCheck[1];	AuliRFIDCheck[11];	AuliRFIDCheck[21];	AuliRFIDCheck[31];	AuliRFIDCheck[41];	AuliRFIDCheck[51];	//...
AuliRFIDCheck[2];	AuliRFIDCheck[12];	AuliRFIDCheck[22];	AuliRFIDCheck[32];	AuliRFIDCheck[42];	AuliRFIDCheck[52];
AuliRFIDCheck[3];	AuliRFIDCheck[13];	AuliRFIDCheck[23];	AuliRFIDCheck[33];	AuliRFIDCheck[43];	AuliRFIDCheck[53];
AuliRFIDCheck[4];	AuliRFIDCheck[14];	AuliRFIDCheck[24];	AuliRFIDCheck[34];	AuliRFIDCheck[44];	AuliRFIDCheck[54];
AuliRFIDCheck[5];	AuliRFIDCheck[15];	AuliRFIDCheck[25];	AuliRFIDCheck[35];	AuliRFIDCheck[45];	AuliRFIDCheck[55];
AuliRFIDCheck[6];	AuliRFIDCheck[16];	AuliRFIDCheck[26];	AuliRFIDCheck[36];	AuliRFIDCheck[46];	AuliRFIDCheck[56];
AuliRFIDCheck[7];	AuliRFIDCheck[17];	AuliRFIDCheck[27];	AuliRFIDCheck[37];	AuliRFIDCheck[47];	AuliRFIDCheck[57];
AuliRFIDCheck[8];	AuliRFIDCheck[18];	AuliRFIDCheck[28];	AuliRFIDCheck[38];	AuliRFIDCheck[48];	AuliRFIDCheck[58];
AuliRFIDCheck[9];	AuliRFIDCheck[19];	AuliRFIDCheck[29];	AuliRFIDCheck[39];	AuliRFIDCheck[49];	AuliRFIDCheck[59];
AuliRFIDCheck[10];	AuliRFIDCheck[20];	AuliRFIDCheck[30];	AuliRFIDCheck[40];	AuliRFIDCheck[50];	AuliRFIDCheck[60];

*)
END_ACTION

ACTION aRFIDCheckWarnings:

(*Brak odczytu RFID przed dozownikami*)
tonRFIDCheckDispencersWarning(IN:= 	(
									(
										(eDispencersPackageState[1].bFormPresent AND (eDispencersPackageState[1].nCardNumber = 0 OR eDispencersPackageState[1].nCardNumber = 999))	OR
										(eDispencersPackageState[2].bFormPresent AND (eDispencersPackageState[2].nCardNumber = 0 OR eDispencersPackageState[2].nCardNumber = 999))	OR 	
										(eDispencersPackageState[3].bFormPresent AND (eDispencersPackageState[3].nCardNumber = 0 OR eDispencersPackageState[3].nCardNumber = 999)) 	OR 
										(eDispencersPackageState[4].bFormPresent AND (eDispencersPackageState[4].nCardNumber = 0 OR eDispencersPackageState[4].nCardNumber = 999))	
										AND NOT bDosingTwoPhases 
									) OR
									(
									(eBeforeDispencer34PackageState2Phase[1].bFormPresent AND eBeforeDispencer34PackageState2Phase[1].nCardNumber = 0) OR
									(eBeforeDispencer34PackageState2Phase[2].bFormPresent AND eBeforeDispencer34PackageState2Phase[2].nCardNumber = 0)
									AND bDosingTwoPhases
									)
								)
								
								AND P00_PackML.tonLongDelayAfterStart.Q AND P00_PackML.fbPMLAuto.ePMLState = Tc3_PackML.E_PMLState.ePMLState_EXECUTE AND
								NOT bRFIDCheckDispencerWarning
								
								, PT:=T#500MS);
							
rttonRFIDCheckDispencerWarning										(CLK:=tonRFIDCheckDispencersWarning.Q, Q=> );
IF rttonRFIDCheckDispencerWarning.Q							THEN	iRFIDCheckDispencerWarning	:=	iRFIDCheckDispencerWarning	+	1;	END_IF;
IF P02_Dispencers.fbDispencersDragRightStation.bCycleDone	THEN	bRFIDCheckDispencerWarning	:= FALSE;								END_IF
(*Koniec Brak odczytu RFID przed dozownikami*)
				

(*Brak odczytu RFID przed waga*)
tonRFIDCheckWeightWarning(IN:= 	(							
										(eWeightPackageState[1].bFormPresent AND eWeightPackageState[1].nCardNumber = 0)	OR
										(eWeightPackageState[2].bFormPresent AND eWeightPackageState[2].nCardNumber = 0)	OR 	
										(eWeightPackageState[3].bFormPresent AND eWeightPackageState[3].nCardNumber = 0) 	OR 
										(eWeightPackageState[4].bFormPresent AND eWeightPackageState[4].nCardNumber = 0)									
								)
								
								AND P00_PackML.tonLongDelayAfterStart.Q AND P00_PackML.fbPMLAuto.ePMLState = Tc3_PackML.E_PMLState.ePMLState_EXECUTE AND
								NOT bRFIDCheckWeightWarning
								
								, PT:=T#500MS);
							
rttonRFIDCheckWeightWarning										(CLK:=tonRFIDCheckWeightWarning.Q, Q=> );
IF rttonRFIDCheckWeightWarning.Q							THEN	iRFIDCheckWeightWarning	:=	iRFIDCheckWeightWarning	+	1;	END_IF;
IF P05_Weight.fbWeightStation.eRunningState = E_WeightLiftStationState.eWeightLiftDown			THEN	bRFIDCheckWeightWarning	:=	FALSE;							END_IF
(*Koniec Brak odczytu RFID przed waga*)


(*Brak odczytu RFID przed zakrecarka*)
tonRFIDCheckBeforeScrewerWarning(IN:= 	(							
										(eUnderScrewerPackageState[1].bFormPresent AND eUnderScrewerPackageState[1].nCardNumber = 0)	OR
										(eUnderScrewerPackageState[2].bFormPresent AND eUnderScrewerPackageState[2].nCardNumber = 0)										
								)
								
								AND P00_PackML.tonLongDelayAfterStart.Q AND P00_PackML.fbPMLAuto.ePMLState = Tc3_PackML.E_PMLState.ePMLState_EXECUTE AND
								NOT bRFIDCheckBeforeScrewerWarning
								
								, PT:=T#500MS);
							
rttonRFIDCheckBeforeScrewerWarning										(CLK:=tonRFIDCheckBeforeScrewerWarning.Q, Q=> );
IF rttonRFIDCheckBeforeScrewerWarning.Q							THEN	iRFIDCheckBeforeScrewerWarning	:=	iRFIDCheckBeforeScrewerWarning	+	1;	END_IF;
IF P10_GripperScrewer.fbGripperScrewersDragStation.bCycleDone	THEN	bRFIDCheckBeforeScrewerWarning	:=	FALSE;									END_IF
(*Koniec Brak odczytu RFID przed zakrecarka*)


(*Brak odczytu RFID za zakrecarka*)
rttonRFIDCheckAfterScrewerWarning	(CLK:=eUnderCorrectCapPackageState[1].bFormPresent, Q=>);
IF rttonRFIDCheckAfterScrewerWarning.Q THEN
	bRFIDCheckAfterScrewerWarning := TRUE;
END_IF
IF bRFIDCheckAfterScrewerWarning AND eUnderCorrectCapPackageState[1].nCardNumber > 0 THEN
	bRFIDCheckAfterScrewerWarning := FALSE;
END_IF
ftRFIDCheckAfterScrewerWarning(CLK:=eUnderCorrectCapPackageState[1].bFormPresent ,CLK=>);			
IF ftRFIDCheckAfterScrewerWarning.Q AND bRFIDCheckAfterScrewerWarning		THEN	
	iRFIDCheckAfterScrewerWarning	:=	iRFIDCheckAfterScrewerWarning	+	1;	
	bRFIDCheckAfterScrewerWarning	:=	FALSE;
END_IF;
(*Koniec Brak odczytu RFID za zakrecarka*)

(*Brak odczytu RFID robot*)
tonRFIDCheckBottleTransferWarning(IN:= 	(							
										(eRobotPackageState[1].bFormPresent AND (eRobotPackageState[1].nCardNumber = 0 OR eRobotPackageState[1].nCardNumber = 999))	OR
										(eRobotPackageState[2].bFormPresent AND (eRobotPackageState[2].nCardNumber = 0 OR eRobotPackageState[2].nCardNumber = 999))										
								)
								AND P00_PackML.iBottleTransferCase = 1
								AND P00_PackML.tonLongDelayAfterStart.Q AND P00_PackML.fbPMLAuto.ePMLState = Tc3_PackML.E_PMLState.ePMLState_EXECUTE AND
								NOT bRFIDCheckBottleTransferWarning
								
								, PT:=T#500MS);
							
rttonRFIDCheckBottleTransferWarning											(CLK:=tonRFIDCheckBottleTransferWarning.Q, Q=> );
IF rttonRFIDCheckBottleTransferWarning.Q							THEN	iRFIDCheckBottleTransferWarning	:=	iRFIDCheckBottleTransferWarning	+	1;	END_IF;
IF P00_PackML.iBottleTransferCase = 3								THEN	bRFIDCheckBottleTransferWarning	:=	FALSE;									END_IF
(*Koniec Brak odczytu RFID robot*)
END_ACTION

ACTION aWriteDataIFM:
tonWriteDataCASE40	(IN:=iWriteDataCASE	=	40,	PT:=T#2S);
IF NOT iWriteDataOn THEN
	iWriteDataCASE							:=	0;
	fbAfterDispencersReader.bReadEnable		:=	TRUE;
	fbAfterDispencersReader.bWriteCmd 		:=	FALSE;
END_IF
CASE iWriteDataCASE OF
	
	0:
		
		fbAfterDispencersReader.diWriteData; // Od ilu zacząć
		IF iWriteDataOn THEN
			fbAfterDispencersReader.bReadEnable		:=	FALSE;
			iWriteDataCASE							:=	iWriteDataCASE	+	10;
		END_IF
		
	10:
		fbAfterDispencersReader.bWriteCmd 		:=	TRUE;
		iWriteDataCASE							:=	iWriteDataCASE	+	10;
		fbAfterDispencersReader.diWriteData;
		
	20:
		IF fbAfterDispencersReader.bWriteCycleEnd 	THEN
			fbAfterDispencersReader.bWriteCmd  	:=	FALSE;
			iWriteDataCASE						:=	iWriteDataCASE	+	10;
		END_IF
		
	30:
		iWriteDataCount	:= iWriteDataCount	+	1;
		
		IF iWriteDataCount	>= 2	THEN
			iWriteDataCount						:=	0;
			fbAfterDispencersReader.diWriteData	:=	fbAfterDispencersReader.diWriteData	+	1;
		END_IF
		
		iWriteDataCASE	:=	iWriteDataCASE	+	10;
		
	40:
		IF NOT fbAfterDispencersReader.bWriteCycleEnd AND tonWriteDataCASE40.Q THEN
			iWriteDataCASE						:=	0;	
		END_IF

END_CASE
END_ACTION

END_PROGRAM

// ---- POUs/FB/FB_WriteRFID.TcPOU
FUNCTION_BLOCK FB_WriteRFID
VAR_INPUT
	bAutoNumber				:BOOL;		
	byFirstByteInput		:BYTE;
	bySecondByteInput		:BYTE;
	byLastByteInput			:BYTE;

	bReset					:BOOL;		//reset licznika
END_VAR
VAR_IN_OUT
	bEnable					:BOOL;		//zalczenie bloku
	byIDtoWrite				:BYTE;		//ID do wczytania
END_VAR


VAR_OUTPUT
	byFirstByteOutput		:BYTE;
	bySecondByteOutput		:BYTE;
	byThirdByteOutput		:BYTE;
	byFourthByteOutput		:BYTE;
	byFifthByteOutput		:BYTE;
	byLastByteOutput		:BYTE;
	bDone					:BOOL;		//informacja o prawidlowym zakoczeniu zapisu
	bError					:BOOL;
	iCounterDone			:INT;		//licznik operacji zapisu zakonczonych sukcesem
END_VAR
VAR
	
	iStep: INT;
	tonDelayError	:TON;
END_VAR

IF bReset THEN
	iCounterDone	:=0;
	iStep := 0;
	byFirstByteOutput := byLastByteOutput := 0;
	bReset := FALSE;
END_IF

CASE iStep OF
	0:  //init	
		IF byFirstByteInput = 129 AND bEnable THEN
			bDone:=FALSE; 
			iStep:=10;
		END_IF
	
	10:  //write command
		bySecondByteOutput 	:= 02;
		byThirdByteOutput	:= 00;
		byFourthByteOutput	:= 00;
		byFifthByteOutput 	:= 01;
		byFirstByteOutput := byLastByteOutput := 01;
	
		IF byFirstByteInput = 163 THEN
			iStep := 20;
		ELSIF NOT byFirstByteInput = 163 AND tonDelayError.Q = TRUE THEN
			iStep := 100;
		END_IF
	
	20: //write data
		IF bAutoNumber THEN
			bySecondByteOutput := byIDtoWrite + INT_TO_BYTE(iCounterDone); 
		ELSE
			bySecondByteOutput := byIDtoWrite;
		END_IF
			
		byFirstByteOutput := byLastByteOutput := 65;
		IF byFirstByteInput = 167 THEN
			iStep := 30;
		ELSIF NOT byFirstByteInput = 167 AND tonDelayError.Q = TRUE THEN
			iStep := 100;
		END_IF
	
	30: //check status
		byFirstByteOutput := byLastByteOutput := 0;
		iCounterDone	:= iCounterDone + 1; 
		bDone			:= TRUE; 	
		IF byFirstByteInput = 128 THEN
			iStep := 0;
			byIDtoWrite		:= byIDtoWrite+1;	
		ELSIF NOT byFirstByteInput = 128 AND tonDelayError.Q = TRUE THEN
			iStep := 100;
		END_IF
		bEnable:=FALSE;
	100: // errors
		bError		:= TRUE;
		



END_CASE

END_FUNCTION_BLOCK

// ---- POUs/FB/FB_WriteRFIDnew.TcPOU
FUNCTION_BLOCK FB_WriteRFIDnew
VAR_INPUT
	bAutoNumber				:BOOL;		
	byFirstByteInput		:BYTE;
	bySecondByteInput		:BYTE;
	byLastByteInput			:BYTE;

	bReset					:BOOL;		//reset licznika
END_VAR
VAR_IN_OUT
	bEnable					:BOOL;		//zalczenie bloku
	byIDtoWrite				:BYTE;		//ID do wczytania
END_VAR


VAR_OUTPUT
	byFirstByteOutput		:BYTE;
	bySecondByteOutput		:BYTE;
	byThirdByteOutput		:BYTE;
	byFourthByteOutput		:BYTE;
	byFifthByteOutput		:BYTE;
	byLastByteOutput		:BYTE;
	bDone					:BOOL;		//informacja o prawidlowym zakoczeniu zapisu
	bError					:BOOL;
	iCounterDone			:INT;		//licznik operacji zapisu zakonczonych sukcesem
END_VAR
VAR
	
	iStep: INT;
	tonDelayError	:TON;
	tonStep0: TON;
	nAutoNumberCount2: INT;
END_VAR

IF bReset THEN
	iCounterDone	:=0;
	iStep := 0;
	byFirstByteOutput := byLastByteOutput := 0;
	bReset := FALSE;
	nAutoNumberCount2:=0;
END_IF

tonStep0(IN:=iStep=0 AND bEnable,PT:=T#500MS);

CASE iStep OF
	0:  //init	
		IF byFirstByteInput = 129 AND tonStep0.Q THEN
			bDone:=FALSE; 
			iStep:=10;
		END_IF
	
	10:  //write command
		bySecondByteOutput 	:= 02;
		byThirdByteOutput	:= 00;
		byFourthByteOutput	:= 00;
		byFifthByteOutput 	:= 01;
		byFirstByteOutput := byLastByteOutput := 01;
	
		IF byFirstByteInput = 163 THEN
			iStep := 20;
		ELSIF NOT byFirstByteInput = 163 AND tonDelayError.Q = TRUE THEN
			iStep := 100;
		END_IF
	
	20: //write data
	
		bySecondByteOutput := byIDtoWrite;
		
		byFirstByteOutput := byLastByteOutput := 65;
		IF byFirstByteInput = 167 THEN
			iStep := 30;
		ELSIF NOT byFirstByteInput = 167 AND tonDelayError.Q = TRUE THEN
			iStep := 100;
		END_IF
	
	30: //check status
		byFirstByteOutput := byLastByteOutput := 0;
		iCounterDone	:= iCounterDone + 1; 
		bDone			:= TRUE; 	
		IF byFirstByteInput = 128 THEN
			iStep := 0;			
			//Liczenie do dwóch i dopiero potem dodaje +1	
			nAutoNumberCount2 := nAutoNumberCount2 + 1;
			IF nAutoNumberCount2 = 2 THEN
				byIDtoWrite			:= byIDtoWrite+1;
				bEnable				:= FALSE;
				nAutoNumberCount2 	:= 0;
			END_IF
			
		ELSIF NOT byFirstByteInput = 128 AND tonDelayError.Q = TRUE THEN
			iStep := 100;
		END_IF
		
	100: // errors
		bError		:= TRUE;
		



END_CASE

END_FUNCTION_BLOCK

// ---- POUs/P02_Dispencers.TcPOU
(*
Nazwa:			P02_Dispencers
Opis:			Stacja dozownikow
Wersja:			v0.1
Data:			2018-10-10
Autor:			DP
Urzadzenia:		
Konfiguracja:	
Info:

*)
PROGRAM P02_Dispencers
VAR_INPUT
	IbDispencer1DropCatcherBackSensor			AT %I*		:BOOL;					//	Czujnik wycofania tacki kropel dozowników
	IbDispencer2DropCatcherBackSensor 			AT %I*		:BOOL;					//	Czujnik wycofania tacki kropel dozowników
	IbDispencer3DropCatcherBackSensor 			AT %I*		:BOOL;					//	Czujnik wycofania tacki kropel dozowników
	IbDispencer4DropCatcherBackSensor 			AT %I*		:BOOL;					//	Czujnik wycofania tacki kropel dozowników
	IbDispencersCatch1SensorValue 				AT %I*		:DINT;					//	Wejscie czujnika otwarcia siłownika chwytania
	IbDispencersCatch2SensorValue				AT %I*		:DINT;					//	Wejscie czujnika otwarcia siłownika chwytania
	IbDispencersCatch3SensorValue				AT %I*		:DINT;					//	Wejscie czujnika otwarcia siłownika chwytania
	IbDispencersCatch4SensorValue				AT %I*		:DINT;					//	Wejscie czujnika otwarcia siłownika chwytania
	IbDispencersDragLeftLeadBefore1UpSensor		AT %I*		:BOOL;					//	Czujnik
	IbDispencersDragLeftLeadAfter1UpSensor		AT %I*		:BOOL;					//	Czujnik
	IbDispencersDragRightLeadBefore1UpSensor	AT %I*		:BOOL;					//	Czujnik
	IbDispencersDragRightLeadAfter1UpSensor		AT %I*		:BOOL;					//	Czujnik
	IbDispencersDragLeftDragUpSensor 			AT %I*		:BOOL;					// 	Czujnik
	IbDispencersDragLeftDragDownSensor 			AT %I*		:BOOL;					// 	Czujnik
	IbDispencersDragRightDragUpSensor 			AT %I*		:BOOL;					// 	Czujnik
	IbDispencersDragRightDragDownSensor 		AT %I*		:BOOL;					// 	Czujnik
	IbDispencersDragLeftDragHomingSensor 		AT %I*		:BOOL;					//	Czujnik bazowania
	IbDispencersDragRightDragHomingSensor 		AT %I*	 	:BOOL;					//	Czujnik bazowania
	IbDispencerAfterCheckFormSensor				AT %I*		:BOOL; 					//	Czujnik po przecionganiu formatek na ukos
	IbDispencer12NoColisionWhenDosingSensor		AT %I*		:BOOL:=TRUE;			//	Czujnik indukcyjny
	IbDispencer34NoColisionWhenDosingSensor		AT %I*		:BOOL:=TRUE;			//	Czujnik indukcyjny
	//EX
	IbTankLevelHighEX									AT %I*:BOOL;
	IbTankLevelLowEX                                    AT %I*:BOOL;
	IbTankLevelExError									AT %I*:BOOL;
END_VAR
VAR
	
	(*******DOZOWNIK 1*********)
	fbDispencer1										: FB_ServoDispencerServoLifter;			//Blok sterujacy dozownikiem nr1
	eDispencer1State									: E_Station; 							// Stan pracy podajnika platynek			
	eDispencer1RunningState								: E_DispencerState; 
	fbDispencer1State									: FB_State;	
	
	tonDispencer1SuckingValveOpenedSensor				: TON;			//Symulacja czujników 
	tonDispencer1DosingValveOpenedSensor				: TON;			//Symulacja czujników 
	tonDispencer1DosingValveClosedSensor				: TON;			//Symulacja czujników 
	tonDispencer1SuckingValveClosedSensor				: TON;
	
	//WEJŚCIA WYJŚCIA SPRZĘTOWE
	//IbDispencer1SuckingValveOpenedSensor AT%I*:BOOL;	(*dok IO-L*)	//Czujnik otwarcia zaworu ssącego dozownika 1
	QbDispencer1DropCatcherValveActuator				:BOOL;			(*Pneu*)		//Otwarcie tacki
	//IbDispencer1SuckingValveClosedSensor AT%I*:BOOL;	(*dok IO-L*)	//Czujnik zamknięcia zaworu ssąceg odozownika 1
	QbDispencer1SuckingValveActuator					:BOOL;				(*Pneu*)		//sterowanie zaworem ssącego (podłaczenie do wyspypneu)
	QbDispencer1DosingValveActuator						:BOOL;				(*Pneu*)		//sterowanie zaworem dozującym (podłaczenie do wyspypneu)
	
	(*******DOZOWNIK 2*********)
	fbDispencer2										: FB_ServoDispencerServoLifter;				//Blok sterujacy dozownikiem nr 1
	eDispencer2State									: E_Station; 							// Stan pracy podajnika platynek			
	eDispencer2RunningState								: E_DispencerState; 
	fbDispencer2State									: FB_State;	
	
	tonDispencer2SuckingValveOpenedSensor				: TON;			//Symulacja czujników 
	tonDispencer2DosingValveOpenedSensor				: TON;			//Symulacja czujników 
	tonDispencer2DosingValveClosedSensor				: TON;			//Symulacja czujników 
	tonDispencer2SuckingValveClosedSensor				: TON;
	
	//WEJŚCIA WYJŚCIA SPRZĘTOWE
	QbDispencer2DropCatcherValveActuator				:BOOL;			(*Pneu*)			//sterowanie tacką kropel(podłaczenie do wyspy pneu)
	//IbDispencer2SuckingValveOpenedSensor AT%I*:BOOL;	(*dok IO-L*)		//Czujnik otwarcia zaworu ssącego dozownika 1
	//IbDispencer2SuckingValveClosedSensor AT%I*:BOOL;	(*dok IO-L*)		//Czujnik zamknięcia zaworu ssącego dozownika 1
	QbDispencer2SuckingValveActuator					:BOOL;				(*Pneu*)			//sterowanie zaworem ssącego(podłaczeniedowyspypneu)
	QbDispencer2DosingValveActuator						:BOOL;				(*Pneu*)			//sterowanie zaworemd ozującym(podłaczeniedowyspypneu)
	QbDispencerDropCatcherSuck							:BOOL;				(*Pneu*)				//Zasysanie płynu z tacek

	(*******DOZOWNIK 3*********)
	fbDispencer3										: FB_ServoDispencerServoLifter;				//Blok sterujacy dozownikiem nr 1
	eDispencer3State									: E_Station; 							// Stan pracy podajnika platynek			
	eDispencer3RunningState								: E_DispencerState; 
	fbDispencer3State									: FB_State;	
	
	tonDispencer3SuckingValveOpenedSensor				: TON;			//Symulacja czujników 
	tonDispencer3DosingValveOpenedSensor				: TON;			//Symulacja czujników 
	tonDispencer3DosingValveClosedSensor				: TON;			//Symulacja czujników 
	tonDispencer3SuckingValveClosedSensor				: TON;
	
	//WEJŚCIA WYJŚCIA SPRZĘTOWE
	QbDispencer3DropCatcherValveActuator				:BOOL;			(*Pneu*)			//Sterowanie tacką kropel(podłaczenie do wyspy pneu)
	//IbDispencer2SuckingValveOpenedSensor AT%I*:BOOL;	(*dok IO-L*)		//Czujnik otwarcia zaworu ssącego dozownika 1
	//IbDispencer2SuckingValveClosedSensor AT%I*:BOOL;	(*dok IO-L*)		//Czujnik zamknięcia zaworu ssącego dozownika 1
	QbDispencer3SuckingValveActuator					:BOOL;				(*Pneu*)			//sterowanie zaworem ssącego(podłaczeniedowyspypneu)
	QbDispencer3DosingValveActuator						:BOOL;				(*Pneu*)			//sterowanie zaworemd ozującym(podłaczeniedowyspypneu)

	(*******DOZOWNIK 4*********)
	fbDispencer4										: FB_ServoDispencerServoLifter;			// Blok sterujacy dozownikiem nr 1
	eDispencer4State									: E_Station; 							// Stan pracy podajnika platynek			
	eDispencer4RunningState								: E_DispencerState; 
	fbDispencer4State									: FB_State;	
	
	tonDispencer4SuckingValveOpenedSensor				: TON;			//Symulacja czujników 
	tonDispencer4DosingValveOpenedSensor				: TON;			//Symulacja czujników 
	tonDispencer4DosingValveClosedSensor				: TON;			//Symulacja czujników 
	tonDispencer4SuckingValveClosedSensor				: TON;
	
	//WEJŚCIA WYJŚCIA SPRZĘTOWE
	QbDispencer4DropCatcherValveActuator				:BOOL;			(*Pneu*)			//sterowanie tacką kropel(podłaczenie do wyspy pneu)
	//IbDispencer2SuckingValveOpenedSensor AT%I*:BOOL;	(*dok IO-L*)		//Czujnik otwarcia zaworu ssącego dozownika 1
	//IbDispencer2SuckingValveClosedSensor AT%I*:BOOL;	(*dok IO-L*)		//Czujnik zamknięcia zaworu ssącego dozownika 1
	QbDispencer4SuckingValveActuator					:BOOL;				(*Pneu*)			//sterowanie zaworem ssącego(podłaczeniedowyspypneu)
	QbDispencer4DosingValveActuator						:BOOL;				(*Pneu*)			//sterowanie zaworemd ozującym(podłaczeniedowyspypneu)
	
	(*******PODNOSNIK TACKI I CHWYTAKA*********)
	fbDispencersCatch1Station							:FB_CatchStationWithSensor;			// Blok stacji chwytaka dozowników
	fbDispencersCatch2Station							:FB_CatchStationWithSensor;			// Blok stacji chwytaka dozowników
	fbDispencersCatch3Station							:FB_CatchStationWithSensor;			// Blok stacji chwytaka dozowników
	fbDispencersCatch4Station							:FB_CatchStationWithSensor;			// Blok stacji chwytaka dozowników
	eDispencersCatch1State								:E_Station; 				// Stan chwytaka stabilizujšcego pod podajnikiem platynek
	eDispencersCatch2State								:E_Station; 				// Stan chwytaka stabilizujšcego pod podajnikiem platynek
	eDispencersCatch3State								:E_Station; 				// Stan chwytaka stabilizujšcego pod podajnikiem platynek
	eDispencersCatch4State								:E_Station; 				// Stan chwytaka stabilizujšcego pod podajnikiem platynek
	eDispencersCatch1RunningState						:E_CatchStationState; 		// Poprzedni stan chwytaka pod podajnikiem nakrętek
	eDispencersCatch2RunningState						:E_CatchStationState; 		// Poprzedni stan chwytaka pod podajnikiem nakrętek
	eDispencersCatch3RunningState						:E_CatchStationState; 		// Poprzedni stan chwytaka pod podajnikiem nakrętek
	eDispencersCatch4RunningState						:E_CatchStationState; 		// Poprzedni stan chwytaka pod podajnikiem nakrętek
	fbDispencersCatch1State								:FB_State;
	fbDispencersCatch2State								:FB_State;
	fbDispencersCatch3State								:FB_State;
	fbDispencersCatch4State								:FB_State;
	
//WEJSCIA I WYJSCIA SPRZETOWE
	QbDispencersCatch1HeightUpCmd 				AT %Q*	:BOOL; 			(*PLC.A17*)		// Wyjście sterujące podnośnikiem chwytaka i tacki dozownika , Silnik w górę
	QbDispencersCatch1HeightDownCmd 			AT %Q*	:BOOL; 		(*PLC.A17*)		// Wyjście sterujące podnośnikiem chwytaka i tacki dozownika, Silnik w dół
	IbDispencersCatch1HeightEncoderPulses 		AT %I*	:BOOL;	(*PLC.A13*)
	
	IbDispencersCatchHeightEncoderSetCDone		AT %I*: BOOL;
	IudiDispencersCatchHeightEncoderCV          AT %I*: UDINT; 
	QbDispencersCatchHeightEncoderSetC 			AT %Q*: BOOL;		
	QudiDispencersCatchHeightEncoderSetCV       AT %Q*: UDINT; 	
	                                            	
	                                            	
	
	
	QbDispencersCatch1Actuator 							:BOOL;					(*Pneu*)		// Wyjście sterujące chwytakiem pod dozownikami
	QbDispencersCatch2Actuator 							:BOOL;					(*Pneu*)		// Wyjście sterujące chwytakiem pod dozownikami
	QbDispencersCatch3Actuator 							:BOOL;					(*Pneu*)		// Wyjście sterujące chwytakiem pod dozownikami
	QbDispencersCatch4Actuator 							:BOOL;					(*Pneu*)		// Wyjście sterujące chwytakiem pod dozownikami

	QbDispencersCatchMaxPressure						:BOOL;				(*Pneu*)			//sterowanie zaworemd ozującym(podłaczeniedowyspypneu)
	
	(*****************SZLABANY*******************)
	fbDispencerGatesStation								:FB_EntranceGatesServo;			// Blok stacji szlabanów 
		
	(*******PRZECIAGANIE**********)
	eDispencersDragLeftStation							: E_Station;
	eDispencersDragLeftRunningStation					: E_DragStationState;
	fbDispencersDragLeftState							: FB_State;
	eDispencersDragRightStation							: E_Station;
	eDispencersDragRightRunningStation					: E_DragStationState;
	fbDispencersDragRightState							: FB_State;	
	fbDispencersDragLeftStation							: FB_FormsDragStepper;	
	fbDispencersDragRightStation						: FB_FormsDragStepper;
	
	//WEJSCIA I WYJSCIA SPRZETOWE
	
	QbDispencersDragLeftDragActuator                   :BOOL;						// Siłownikiem przeciągania (1 faza)
	
	QbDispencersDragLeftLeadBefore1Actuator          :BOOL;							// Siłownikiem prowadzenia przed 1(1 faza)
	QbDispencersDragLeftLeadAfter1Actuator          :BOOL;							// Siłownikiem prowadzenia przed 1(1 faza)
	
	QbDispencersDragRightDragActuator                  :BOOL;						// Siłownikiem przeciągania (1 faza)
	
	QbDispencersDragRightLeadBefore1Actuator          :BOOL;						// Siłownikiem prowadzenia przed 2(1 faza)	
	QbDispencersDragRightLeadAfter1Actuator          :BOOL;							// Siłownikiem prowadzenia przed 1(1 faza)
		
	(**********ZBIORNIKI**************)
	//Zbiornik
	IbTank1LevelLow 							 AT %I* :BOOL; 				(*PLC.A8*)	// Niski poziom masy w zbiorniku
	IbTank2LevelLow 							 AT %I* :BOOL; 				(*PLC.A8*)	// Niski poziom masy w zbiorniku
	QbTank1LevelSensorCalibration 			     AT %Q* :BOOL;  (*PLC.A20*)	// Kalibracja czujnika poziomu leja nr 1
	QbTank2LevelSensorCalibration 				 AT %Q* :BOOL;  (*PLC.A20*)	// Kalibracja czujnika poziomu leja nr 2
	
	
	QbTank1Pressure								 AT %Q* :BOOL;						(*Pneu*)	// Ciśnienie w zbiorniku nr 1
	bTank1LevelLow                                      :BOOL;									// Sygnały sterujące pompy 1 zależnie od ich odwrócenia
	bTank2LevelLow										:BOOL;									// Sygnały sterujące pompy 2 zależnie od ich odwrócenia
	
	//Pompa podająca
	QbTank1PumpStart 							AT %Q*	:BOOL;		(*PLC.A21*)	//Załączenie pompy masy do zbiornika
	QbTank2PumpStart 							AT %Q*	:BOOL;		(*PLC.A21*)	//Załączenie pompy masy do zbiornika
	QbTank3PumpStart 							AT %Q*	:BOOL;		(*PLC.A21*)	//Załączenie pompy masy do zbiornika
	QbTank4PumpStart 							AT %Q*	:BOOL;		(*PLC.A21*)	//Załączenie pompy masy do zbiornika
	IbTank1PumpFuseOK 							AT %I*  :BOOL; 				//Potwierdzenie z zabezpieczenia pompy 1 - OK
	IbTank2PumpFuseOK 							AT %I*  :BOOL; 				//Potwierdzenie z zabezpieczenia pompy 2 - OK
	IbTank3PumpFuseOK 							AT %I*  :BOOL; 				//Potwierdzenie z zabezpieczenia pompy 2 - OK
	IbTank4PumpFuseOK 							AT %I*  :BOOL; 				//Potwierdzenie z zabezpieczenia pompy 2 - OK
		
	(*GRZAŁKA ZBIORNIKA*)
	fbTankHeating										: FB_TankHeating;	
	eTankHeatingState									: E_Station; 					// Stan pracy grzania
	eTankHeatingRunningState							: E_MassHeatingState; 			// Stan pracy grzania
	fbTankHeatingState									: FB_State;
		
	//WEJŚĆIA I WYJŚĆIA SPRZĘTOWE		
	QbTankHeatingPWMOut							AT %Q* :BOOL; 					// Wyjście sterujące temperaturą grzałki
	AInTankHeatingTempCVSensor 					AT %I* :INT; 			// Wartość aktualnej temperatury grzałki
	IbTankHeatingTempSensorFailure 				AT %I* :BOOL;  		// Informacja o uszkodzeniu czujnika temperatury grzałki	
	
	//Mieszadło zbiornika
	IbFuseTankMixerEngineOK						AT %I* :BOOL;	(*PLC.A7*)	//Bezpiecznik silnika mieszadła OK
	IbFuseTankMixerEngineWorking				AT %I* :BOOL;	{warning 'oprogramowac nowy sygnał mieszadla'}			//Potwierdzenie pracy silnika mieszadła OK	
	QbTank1MixerStart 							AT %Q* :BOOL;			(*PLC.A20*)	//Załączenie mieszadła masy do zbiornika
	
	// Zezwolenie na pracę mieszadła zbiornikowego
	tonTank1LevelSensor									: TON;
	
	tofTank2LevelSensor									: TOF;
	tonTank2LevelSensor									: TON;
	
	tonTank1LevelWarning	   							: TON;
	tonTank2LevelWarning	   							: TON;
	
	tonTank1EmptyAlarm									: TON;
	tonTank2EmptyAlarm									: TON;
	rtDispencer1DoseDone								: R_TRIG;
	rtDispencer2DoseDone								: R_TRIG;
	
	tonTankLevelSensorCalibrationLight					: TON;
	tonTankLevelSensorCalibrationDark					: TON;
	
	(**********OSLONA DOZOWNIKOW*************)	
	
	nCalibrationDialog								 	: INT;

	TimerDispencer1Enable								: TOF;
	TimerDispencer2Enable								: TOF;
	TimerDispencer3Enable								: TOF;
	TimerDispencer4Enable								: TOF;		
	
	(*Wykres dozowania*)
	fbDosingChart1										: FB_WriteDataToArrayString;
	fbDosingChart2										: FB_WriteDataToArrayString;
	fbDosingChart3										: FB_WriteDataToArrayString;
	fbDosingChart4										: FB_WriteDataToArrayString;
	fbDosingStChart1									: FB_WriteDataToArrayOfArrays;
	fbDosingStChart2									: FB_WriteDataToArrayOfArrays;
	fbDosingStChart3									: FB_WriteDataToArrayOfArrays;
	fbDosingStChart4									: FB_WriteDataToArrayOfArrays;
	nChartCycleTime										: INT;
	tDelayDispencerValve								: TIME;

	rtEnable											: R_TRIG;

	fbDropCatcherSuck									: FB_Blink_AS;
	nDose1Counter										: INT;
	nDose2Counter										: INT;
	nDose1CounterWhenLowLevel							: INT;
	nDose2CounterWhenLowLevel							: INT;	
	nDoseCounter1										: INT;
	nDoseCounter2										: INT;	
	// Czujnik poziomu masy przewodząco pojmenościowy LiquiPoint FTW33
	// Zmienne akcji ACT_ConductiveMassSensor
	
	bTank1LevelLowConductiveSensor						: BOOL;
	bTank1SensorDiagnosis								: BOOL;     // Diagnostyka czujnika
	IusiTank1SensorValue0						AT%I*	: USINT;
	IusiTank1SensorValue1						AT%I*	: USINT;
	IusiTank1SensorValue2						AT%I*	: USINT;
	IusiTank1SensorValue3						AT%I*	: USINT;
	IusiTank1SensorDiagnosis					AT%I*	: USINT;
    iTank1Sensor1Value									: INT;	                         
	tonTank1LevelLowConductiveSensor					: TON;
	iTank1Sensor1ValueTemp								: INT;	
	
